C09129=1221.568,302.817,-67.481,-176.404,6.935,148.235
C09130=1221.564,303.066,-67.511,-176.401,6.937,148.235
C09131=1221.559,303.313,-67.540,-176.399,6.940,148.235
C09132=1221.555,303.561,-67.570,-176.397,6.942,148.235
C09133=1221.551,303.809,-67.599,-176.395,6.944,148.235
C09134=1221.546,304.058,-67.629,-176.392,6.947,148.235
C09135=1221.542,304.306,-67.659,-176.390,6.950,148.235
C09136=1221.538,304.554,-67.688,-176.387,6.953,148.235
C09137=1221.533,304.803,-67.718,-176.385,6.955,148.235
C09138=1221.529,305.051,-67.747,-176.383,6.957,148.235
C09139=1221.525,305.299,-67.778,-176.380,6.960,148.235
C09140=1221.520,305.547,-67.807,-176.378,6.962,148.235
C09141=1221.516,305.795,-67.837,-176.376,6.965,148.235
C09142=1221.512,306.044,-67.866,-176.373,6.968,148.235
C09143=1221.508,306.291,-67.896,-176.371,6.970,148.235
C09144=1221.503,306.540,-67.926,-176.369,6.973,148.235
C09145=1221.499,306.788,-67.956,-176.366,6.975,148.235
C09146=1221.495,307.036,-67.985,-176.364,6.977,148.234
C09147=1221.491,307.284,-68.016,-176.362,6.980,148.234
C09148=1221.486,307.533,-68.046,-176.360,6.983,148.234
C09149=1221.482,307.781,-68.075,-176.357,6.986,148.234
C09150=1221.478,308.029,-68.104,-176.355,6.988,148.234
C09151=1221.473,308.277,-68.135,-176.353,6.990,148.234
C09152=1221.469,308.525,-68.165,-176.350,6.993,148.234
C09153=1221.465,308.774,-68.194,-176.348,6.995,148.234
C09154=1221.460,309.022,-68.225,-176.346,6.998,148.234
C09155=1221.456,309.270,-68.254,-176.343,7.001,148.234
C09156=1221.452,309.517,-68.285,-176.341,7.003,148.234
C09157=1221.447,309.766,-68.315,-176.338,7.006,148.234
C09158=1221.443,310.014,-68.344,-176.336,7.008,148.234
C09159=1221.439,310.262,-68.374,-176.334,7.010,148.234
C09160=1221.434,310.511,-68.404,-176.332,7.013,148.234
C09161=1221.430,310.758,-68.434,-176.329,7.016,148.234
C09162=1221.426,311.006,-68.464,-176.327,7.019,148.234
C09163=1221.422,311.256,-68.494,-176.325,7.021,148.234
C09164=1221.418,311.503,-68.524,-176.323,7.023,148.234
C09165=1221.413,311.752,-68.554,-176.320,7.026,148.234
C09166=1221.409,312.000,-68.585,-176.318,7.028,148.234
C09167=1221.405,312.248,-68.614,-176.316,7.032,148.234
C09168=1221.400,312.496,-68.645,-176.313,7.034,148.234
C09169=1221.396,312.743,-68.675,-176.311,7.036,148.234
C09170=1221.391,312.992,-68.705,-176.309,7.039,148.234
C09171=1221.388,313.240,-68.735,-176.307,7.041,148.234
C09172=1221.383,313.488,-68.765,-176.304,7.044,148.234
C09173=1221.379,313.737,-68.796,-176.302,7.047,148.234
C09174=1221.375,313.985,-68.826,-176.300,7.049,148.234
C09175=1221.371,314.233,-68.856,-176.298,7.052,148.234
C09176=1221.367,314.480,-68.886,-176.295,7.054,148.234
C09177=1221.362,314.729,-68.916,-176.293,7.058,148.234
C09178=1221.357,315.005,-68.951,-176.291,7.060,148.234
C09179=1221.353,315.281,-68.984,-176.288,7.063,148.234
C09180=1221.348,315.557,-69.018,-176.285,7.066,148.234
C09181=1221.343,315.832,-69.050,-176.283,7.069,148.234
C09182=1221.339,316.081,-69.082,-176.281,7.071,148.234
C09183=1221.334,316.329,-69.112,-176.278,7.074,148.234
C09184=1221.330,316.577,-69.142,-176.276,7.077,148.234
C09185=1221.326,316.825,-69.173,-176.274,7.079,148.234
C09186=1221.322,317.073,-69.203,-176.271,7.082,148.234
C09187=1221.317,317.321,-69.233,-176.269,7.084,148.234
C09188=1221.313,317.570,-69.263,-176.267,7.087,148.234
C09189=1221.309,317.818,-69.294,-176.265,7.090,148.234
C09190=1221.305,318.065,-69.324,-176.262,7.093,148.234
C09191=1221.300,318.313,-69.355,-176.260,7.095,148.234
C09192=1221.295,318.562,-69.385,-176.258,7.097,148.234
C09193=1221.292,318.810,-69.416,-176.256,7.101,148.234
C09194=1221.288,319.058,-69.446,-176.254,7.103,148.234
C09195=1221.283,319.306,-69.477,-176.251,7.106,148.234
C09196=1221.279,319.554,-69.507,-176.249,7.108,148.234
C09197=1221.275,319.802,-69.538,-176.247,7.111,148.234
C09198=1221.271,320.051,-69.568,-176.245,7.114,148.234
C09199=1221.266,320.298,-69.599,-176.243,7.116,148.234
C09200=1221.262,320.546,-69.629,-176.240,7.119,148.234
C09201=1221.258,320.795,-69.660,-176.238,7.121,148.234
C09202=1221.254,321.043,-69.691,-176.236,7.124,148.234
C09203=1221.249,321.291,-69.721,-176.234,7.127,148.234
C09204=1221.245,321.538,-69.752,-176.232,7.129,148.234
C09205=1221.241,321.787,-69.783,-176.229,7.132,148.235
C09206=1221.237,322.035,-69.813,-176.227,7.134,148.234
C09207=1221.232,322.283,-69.844,-176.225,7.138,148.234
C09208=1221.228,322.531,-69.874,-176.223,7.140,148.235
C09209=1221.224,322.779,-69.906,-176.221,7.142,148.235
C09210=1221.220,323.027,-69.936,-176.218,7.145,148.235
C09211=1221.216,323.275,-69.966,-176.217,7.148,148.235
C09212=1221.212,323.524,-69.998,-176.214,7.151,148.235
C09213=1221.207,323.771,-70.028,-176.212,7.153,148.235
C09214=1221.202,324.019,-70.059,-176.210,7.156,148.235
C09215=1221.199,324.268,-70.090,-176.207,7.159,148.235
C09216=1221.195,324.516,-70.120,-176.205,7.161,148.235
C09217=1221.190,324.764,-70.151,-176.203,7.164,148.235
C09218=1221.186,325.012,-70.182,-176.201,7.166,148.235
C09219=1221.181,325.260,-70.213,-176.198,7.170,148.235
C09220=1221.178,325.507,-70.244,-176.197,7.172,148.235
C09221=1221.174,325.756,-70.275,-176.195,7.174,148.235
C09222=1221.169,326.004,-70.306,-176.192,7.178,148.235
C09223=1221.165,326.252,-70.337,-176.190,7.180,148.235
C09224=1221.161,326.501,-70.368,-176.188,7.183,148.235
C09225=1221.157,326.748,-70.398,-176.186,7.185,148.236
C09226=1221.152,326.996,-70.429,-176.184,7.188,148.235
C09227=1221.148,327.244,-70.461,-176.182,7.191,148.236
C09228=1221.144,327.492,-70.491,-176.180,7.193,148.236
C09229=1221.139,327.740,-70.522,-176.177,7.196,148.236
C09230=1221.135,327.989,-70.553,-176.175,7.199,148.236
C09231=1221.131,328.236,-70.585,-176.173,7.202,148.236
C09232=1221.127,328.485,-70.616,-176.171,7.204,148.236
C09233=1221.122,328.733,-70.647,-176.169,7.207,148.236
C09234=1221.119,328.980,-70.677,-176.167,7.210,148.236
C09235=1221.115,329.228,-70.709,-176.165,7.212,148.236
C09236=1221.110,329.476,-70.739,-176.163,7.216,148.236
C09237=1221.105,329.724,-70.770,-176.160,7.218,148.236
C09238=1221.102,329.972,-70.802,-176.159,7.220,148.237
C09239=1221.097,330.220,-70.833,-176.156,7.223,148.237
C09240=1221.093,330.469,-70.864,-176.154,7.226,148.237
C09241=1221.089,330.716,-70.895,-176.152,7.229,148.237
C09242=1221.085,330.965,-70.926,-176.150,7.231,148.237
C09243=1221.080,331.212,-70.958,-176.148,7.234,148.237
C09244=1221.076,331.460,-70.989,-176.146,7.237,148.237
C09245=1221.072,331.709,-71.020,-176.144,7.239,148.237
C09246=1221.067,331.956,-71.051,-176.142,7.243,148.237
C09247=1221.063,332.205,-71.082,-176.139,7.245,148.237
C09248=1221.059,332.452,-71.114,-176.137,7.248,148.237
C09249=1221.055,332.701,-71.145,-176.135,7.250,148.237
C09250=1221.051,332.948,-71.177,-176.134,7.253,148.238
C09251=1221.047,333.197,-71.208,-176.131,7.256,148.238
C09252=1221.042,333.444,-71.239,-176.129,7.258,148.238
C09253=1221.038,333.693,-71.270,-176.127,7.262,148.238
C09254=1221.034,333.940,-71.302,-176.125,7.264,148.238
C09255=1221.030,334.188,-71.333,-176.123,7.267,148.238
C09256=1221.026,334.436,-71.364,-176.121,7.270,148.238
C09257=1221.021,334.684,-71.395,-176.119,7.272,148.238
C09258=1221.017,334.933,-71.428,-176.117,7.276,148.239
C09259=1221.012,335.181,-71.458,-176.115,7.278,148.238
C09260=1221.008,335.429,-71.490,-176.113,7.280,148.239
C09261=1221.004,335.677,-71.521,-176.111,7.284,148.239
C09262=1221.000,335.925,-71.553,-176.109,7.286,148.239
C09263=1220.996,336.172,-71.584,-176.107,7.289,148.239
C09264=1220.992,336.421,-71.615,-176.105,7.291,148.239
C09265=1220.988,336.669,-71.647,-176.103,7.294,148.239
C09266=1220.984,336.916,-71.679,-176.101,7.297,148.239
C09267=1220.979,337.165,-71.710,-176.099,7.300,148.239
C09268=1220.975,337.412,-71.742,-176.096,7.303,148.240
C09269=1220.971,337.660,-71.774,-176.095,7.305,148.240
C09270=1220.966,337.908,-71.805,-176.093,7.308,148.240
C09271=1220.963,338.156,-71.836,-176.090,7.311,148.240
C09272=1220.958,338.404,-71.868,-176.089,7.314,148.240
C09273=1220.954,338.653,-71.900,-176.087,7.317,148.240
C09274=1220.949,338.900,-71.931,-176.085,7.319,148.240
C09275=1220.946,339.148,-71.963,-176.083,7.322,148.241
C09276=1220.942,339.396,-71.995,-176.081,7.325,148.241
C09277=1220.937,339.644,-72.026,-176.079,7.328,148.241
C09278=1220.933,339.892,-72.058,-176.076,7.331,148.241
C09279=1220.929,340.140,-72.089,-176.075,7.333,148.241
C09280=1220.925,340.388,-72.121,-176.073,7.336,148.241
C09281=1220.921,340.635,-72.153,-176.071,7.339,148.242
C09282=1220.915,340.913,-72.188,-176.068,7.342,148.242
C09283=1220.911,341.191,-72.224,-176.067,7.345,148.242
C09284=1220.907,341.469,-72.259,-176.064,7.348,148.242
C09285=1220.901,341.747,-72.295,-176.062,7.351,148.242
C09286=1220.897,341.995,-72.327,-176.060,7.353,148.242
C09287=1220.894,342.243,-72.359,-176.058,7.357,148.242
C09288=1220.889,342.491,-72.391,-176.056,7.359,148.243
C09289=1220.885,342.739,-72.423,-176.055,7.362,148.243
C09290=1220.881,342.986,-72.454,-176.053,7.365,148.243
C09291=1220.876,343.234,-72.486,-176.050,7.367,148.243
C09292=1220.872,343.483,-72.518,-176.048,7.371,148.243
C09293=1220.868,343.730,-72.549,-176.047,7.373,148.243
C09294=1220.864,343.979,-72.582,-176.045,7.376,148.244
C09295=1220.860,344.227,-72.613,-176.043,7.379,148.244
C09296=1220.856,344.474,-72.645,-176.041,7.382,148.244
C09297=1220.851,344.723,-72.677,-176.040,7.384,148.244
C09298=1220.847,344.971,-72.709,-176.037,7.388,148.244
C09299=1220.842,345.218,-72.741,-176.035,7.390,148.244
C09300=1220.839,345.466,-72.773,-176.033,7.393,148.245
C09301=1220.835,345.714,-72.805,-176.031,7.396,148.245
C09302=1220.830,345.962,-72.837,-176.030,7.398,148.245
C09303=1220.826,346.210,-72.869,-176.028,7.402,148.245
C09304=1220.822,346.458,-72.902,-176.026,7.404,148.245
C09305=1220.818,346.705,-72.933,-176.024,7.407,148.245
C09306=1220.814,346.953,-72.965,-176.022,7.410,148.246
C09307=1220.810,347.201,-72.998,-176.020,7.413,148.246
C09308=1220.805,347.449,-73.029,-176.019,7.415,148.246
C09309=1220.801,347.697,-73.062,-176.017,7.418,148.246
C09310=1220.797,347.945,-73.094,-176.015,7.421,148.246
C09311=1220.792,348.193,-73.126,-176.013,7.424,148.247
C09312=1220.788,348.441,-73.157,-176.011,7.427,148.247
C09313=1220.784,348.689,-73.191,-176.010,7.429,148.247
C09314=1220.781,348.937,-73.222,-176.007,7.433,148.247
C09315=1220.775,349.184,-73.254,-176.006,7.435,148.247
C09316=1220.772,349.432,-73.286,-176.004,7.438,148.248
C09317=1220.767,349.681,-73.319,-176.002,7.441,148.248
C09318=1220.764,349.928,-73.351,-176.000,7.444,148.248
C09319=1220.759,350.176,-73.383,-175.999,7.446,148.248
C09320=1220.755,350.424,-73.415,-175.996,7.450,148.248
C09321=1220.751,350.672,-73.448,-175.995,7.452,148.249
C09322=1220.747,350.920,-73.480,-175.993,7.455,148.249
C09323=1220.742,351.167,-73.512,-175.991,7.458,148.249
C09324=1220.739,351.415,-73.544,-175.989,7.460,148.249
C09325=1220.734,351.664,-73.577,-175.988,7.463,148.249
C09326=1220.730,351.911,-73.610,-175.986,7.466,148.250
C09327=1220.726,352.159,-73.641,-175.984,7.469,148.250
C09328=1220.721,352.407,-73.674,-175.983,7.472,148.250
C09329=1220.718,352.654,-73.706,-175.981,7.475,148.250
C09330=1220.713,352.903,-73.739,-175.979,7.478,148.251
C09331=1220.710,353.151,-73.771,-175.977,7.480,148.251
C09332=1220.705,353.398,-73.803,-175.975,7.483,148.251
C09333=1220.700,353.646,-73.836,-175.973,7.486,148.251
C09334=1220.697,353.894,-73.868,-175.972,7.489,148.252
C09335=1220.693,354.142,-73.901,-175.970,7.492,148.252
C09336=1220.688,354.390,-73.933,-175.968,7.495,148.252
C09337=1220.684,354.637,-73.965,-175.967,7.497,148.252
C09338=1220.680,354.885,-73.998,-175.965,7.500,148.252
C09339=1220.676,355.133,-74.030,-175.963,7.503,148.253
C09340=1220.672,355.381,-74.063,-175.962,7.506,148.253
C09341=1220.667,355.629,-74.095,-175.960,7.508,148.253
C09342=1220.664,355.877,-74.128,-175.958,7.512,148.253
C09343=1220.659,356.125,-74.160,-175.956,7.514,148.254
C09344=1220.655,356.372,-74.193,-175.955,7.517,148.254
C09345=1220.651,356.620,-74.225,-175.953,7.521,148.254
C09346=1220.647,356.868,-74.258,-175.951,7.523,148.254
C09347=1220.643,357.116,-74.291,-175.950,7.526,148.255
C09348=1220.638,357.364,-74.324,-175.949,7.528,148.255
C09349=1220.635,357.612,-74.356,-175.946,7.532,148.255
C09350=1220.630,357.859,-74.388,-175.945,7.534,148.255
C09351=1220.626,358.107,-74.421,-175.943,7.537,148.256
C09352=1220.622,358.355,-74.453,-175.941,7.540,148.256
C09353=1220.618,358.603,-74.486,-175.940,7.543,148.256
C09354=1220.614,358.851,-74.519,-175.938,7.546,148.257
C09355=1220.609,359.099,-74.552,-175.937,7.548,148.257
C09356=1220.606,359.346,-74.585,-175.935,7.552,148.257
C09357=1220.602,359.595,-74.617,-175.933,7.554,148.257
C09358=1220.597,359.842,-74.650,-175.932,7.557,148.258
C09359=1220.592,360.090,-74.682,-175.930,7.560,148.258
C09360=1220.588,360.338,-74.715,-175.928,7.563,148.258
C09361=1220.585,360.585,-74.748,-175.927,7.566,148.258
C09362=1220.580,360.833,-74.780,-175.925,7.568,148.259
C09363=1220.576,361.081,-74.814,-175.924,7.571,148.259
C09364=1220.572,361.329,-74.847,-175.922,7.574,148.259
C09365=1220.568,361.577,-74.880,-175.921,7.577,148.260
C09366=1220.564,361.825,-74.912,-175.919,7.580,148.260
C09367=1220.560,362.072,-74.945,-175.918,7.583,148.260
C09368=1220.556,362.320,-74.978,-175.916,7.586,148.261
C09369=1220.552,362.568,-75.011,-175.914,7.588,148.261
C09370=1220.547,362.816,-75.044,-175.913,7.591,148.261
C09371=1220.543,363.064,-75.077,-175.911,7.594,148.261
C09372=1220.540,363.311,-75.109,-175.910,7.597,148.262
C09373=1220.536,363.559,-75.143,-175.908,7.600,148.262
C09374=1220.531,363.807,-75.175,-175.907,7.603,148.262
C09375=1220.527,364.054,-75.208,-175.905,7.605,148.262
C09376=1220.522,364.302,-75.241,-175.904,7.608,148.263
C09377=1220.518,364.550,-75.274,-175.903,7.611,148.263
C09378=1220.514,364.798,-75.307,-175.900,7.614,148.264
C09379=1220.510,365.046,-75.340,-175.899,7.617,148.264
C09380=1220.506,365.293,-75.372,-175.898,7.620,148.264
C09381=1220.502,365.541,-75.405,-175.896,7.622,148.264
C09382=1220.498,365.789,-75.439,-175.895,7.625,148.265
C09383=1220.494,366.037,-75.472,-175.893,7.629,148.265
C09384=1220.490,366.284,-75.505,-175.891,7.631,148.265
C09385=1220.486,366.532,-75.538,-175.890,7.634,148.266
C09386=1220.481,366.813,-75.575,-175.889,7.637,148.266
C09387=1220.477,367.093,-75.613,-175.887,7.640,148.266
C09388=1220.472,367.372,-75.650,-175.885,7.644,148.267
C09389=1220.468,367.652,-75.688,-175.884,7.647,148.267
C09390=1220.463,367.900,-75.720,-175.883,7.649,148.268
C09391=1220.459,368.148,-75.753,-175.881,7.652,148.268
C09392=1220.455,368.396,-75.787,-175.879,7.656,148.268
C09393=1220.451,368.643,-75.820,-175.878,7.658,148.269
C09394=1220.447,368.891,-75.853,-175.877,7.661,148.269
C09395=1220.442,369.139,-75.886,-175.875,7.664,148.269
C09396=1220.438,369.386,-75.919,-175.874,7.667,148.270
C09397=1220.434,369.634,-75.952,-175.873,7.669,148.270
C09398=1220.430,369.882,-75.985,-175.871,7.672,148.270
C09399=1220.426,370.130,-76.019,-175.870,7.675,148.271
C09400=1220.422,370.377,-76.053,-175.869,7.678,148.271
C09401=1220.418,370.624,-76.086,-175.867,7.680,148.271
C09402=1220.414,370.872,-76.119,-175.866,7.683,148.272
C09403=1220.410,371.120,-76.152,-175.865,7.687,148.272
C09404=1220.405,371.368,-76.185,-175.863,7.689,148.272
C09405=1220.401,371.616,-76.219,-175.862,7.692,148.273
C09406=1220.397,371.864,-76.252,-175.861,7.695,148.273
C09407=1220.393,372.112,-76.286,-175.859,7.698,148.273
C09408=1220.389,372.360,-76.319,-175.858,7.700,148.274
C09409=1220.385,372.607,-76.352,-175.857,7.703,148.274
C09410=1220.381,372.854,-76.386,-175.856,7.706,148.275
C09411=1220.377,373.102,-76.419,-175.854,7.709,148.275
C09412=1220.373,373.350,-76.452,-175.853,7.711,148.275
C09413=1220.368,373.598,-76.485,-175.852,7.714,148.276
C09414=1220.364,373.845,-76.518,-175.851,7.717,148.276
C09415=1220.359,374.093,-76.552,-175.849,7.720,148.276
C09416=1220.356,374.341,-76.586,-175.848,7.723,148.277
C09417=1220.352,374.589,-76.620,-175.847,7.726,148.277
C09418=1220.348,374.837,-76.653,-175.846,7.728,148.277
C09419=1220.344,375.084,-76.686,-175.845,7.731,148.278
C09420=1220.340,375.332,-76.719,-175.843,7.734,148.278
C09421=1220.336,375.579,-76.753,-175.842,7.736,148.278
C09422=1220.331,375.827,-76.787,-175.841,7.739,148.279
C09423=1220.327,376.075,-76.820,-175.840,7.742,148.279
C09424=1220.323,376.323,-76.853,-175.838,7.745,148.280
C09425=1220.319,376.571,-76.887,-175.837,7.748,148.280
C09426=1220.315,376.818,-76.920,-175.836,7.751,148.280
C09427=1220.311,377.066,-76.953,-175.835,7.753,148.281
C09428=1220.307,377.313,-76.988,-175.834,7.755,148.281
C09429=1220.302,377.561,-77.021,-175.833,7.758,148.282
C09430=1220.298,377.809,-77.054,-175.832,7.761,148.282
C09431=1220.295,378.057,-77.088,-175.831,7.764,148.282
C09432=1220.291,378.304,-77.122,-175.829,7.767,148.283
C09433=1220.286,378.552,-77.155,-175.828,7.769,148.283
C09434=1220.282,378.800,-77.189,-175.827,7.772,148.284
C09435=1220.278,379.047,-77.222,-175.826,7.775,148.284
C09436=1220.274,379.295,-77.256,-175.825,7.778,148.284
C09437=1220.270,379.543,-77.290,-175.824,7.781,148.285
C09438=1220.266,379.791,-77.324,-175.823,7.783,148.285
C09439=1220.262,380.039,-77.357,-175.822,7.786,148.285
C09440=1220.258,380.286,-77.391,-175.821,7.789,148.286
C09441=1220.253,380.534,-77.424,-175.820,7.791,148.286
C09442=1220.249,380.781,-77.458,-175.819,7.794,148.287
C09443=1220.246,381.029,-77.492,-175.817,7.797,148.287
C09444=1220.241,381.277,-77.525,-175.816,7.800,148.288
C09445=1220.237,381.524,-77.559,-175.816,7.802,148.288
C09446=1220.233,381.772,-77.593,-175.814,7.805,148.288
C09447=1220.229,382.019,-77.626,-175.813,7.808,148.289
C09448=1220.225,382.268,-77.660,-175.812,7.810,148.289
C09449=1220.221,382.515,-77.694,-175.811,7.813,148.290
C09450=1220.217,382.763,-77.728,-175.811,7.815,148.290
C09451=1220.212,383.010,-77.762,-175.810,7.818,148.291
C09452=1220.209,383.259,-77.796,-175.808,7.821,148.291
C09453=1220.205,383.506,-77.829,-175.807,7.824,148.291
C09454=1220.200,383.754,-77.863,-175.807,7.826,148.292
C09455=1220.196,384.001,-77.897,-175.805,7.829,148.292
C09456=1220.192,384.249,-77.930,-175.805,7.832,148.293
C09457=1220.188,384.497,-77.965,-175.803,7.835,148.293
C09458=1220.184,384.745,-77.998,-175.802,7.837,148.293
C09459=1220.180,384.992,-78.032,-175.802,7.839,148.294
C09460=1220.175,385.240,-78.066,-175.800,7.842,148.294
C09461=1220.172,385.487,-78.100,-175.800,7.845,148.295
C09462=1220.168,385.735,-78.134,-175.799,7.847,148.295
C09463=1220.163,385.983,-78.168,-175.798,7.850,148.296
C09464=1220.159,386.230,-78.202,-175.797,7.853,148.296
C09465=1220.155,386.478,-78.236,-175.796,7.856,148.297
C09466=1220.151,386.726,-78.269,-175.795,7.858,148.297
C09467=1220.147,386.973,-78.303,-175.794,7.861,148.297
C09468=1220.142,387.221,-78.337,-175.793,7.864,148.298
C09469=1220.139,387.469,-78.371,-175.793,7.866,148.298
C09470=1220.134,387.717,-78.405,-175.792,7.869,148.299
C09471=1220.131,387.964,-78.439,-175.790,7.872,148.299
C09472=1220.127,388.211,-78.473,-175.790,7.874,148.299
C09473=1220.122,388.460,-78.507,-175.789,7.877,148.300
C09474=1220.119,388.707,-78.541,-175.788,7.880,148.300
C09475=1220.114,388.954,-78.575,-175.787,7.881,148.301
C09476=1220.111,389.202,-78.609,-175.786,7.884,148.301
C09477=1220.106,389.450,-78.643,-175.785,7.887,148.302
C09478=1220.102,389.697,-78.677,-175.785,7.889,148.302
C09479=1220.099,389.945,-78.711,-175.783,7.892,148.302
C09480=1220.094,390.193,-78.745,-175.783,7.894,148.303
C09481=1220.090,390.440,-78.779,-175.782,7.897,148.303
C09482=1220.086,390.687,-78.813,-175.781,7.900,148.304
C09483=1220.082,390.936,-78.847,-175.781,7.902,148.304
C09484=1220.077,391.183,-78.881,-175.780,7.905,148.305
C09485=1220.074,391.430,-78.915,-175.779,7.907,148.305
C09486=1220.070,391.678,-78.950,-175.778,7.910,148.306
C09487=1220.066,391.926,-78.983,-175.777,7.913,148.306
C09488=1220.061,392.174,-79.018,-175.776,7.915,148.306
C09489=1220.058,392.421,-79.052,-175.776,7.918,148.307
C09490=1220.053,392.703,-79.091,-175.774,7.921,148.307
C09491=1220.048,392.985,-79.130,-175.774,7.923,148.308
C09492=1220.044,393.267,-79.169,-175.773,7.926,148.308
C09493=1220.039,393.549,-79.207,-175.772,7.929,148.309
C09494=1220.035,393.796,-79.242,-175.771,7.932,148.309
C09495=1220.031,394.044,-79.276,-175.771,7.934,148.310
C09496=1220.027,394.291,-79.310,-175.770,7.937,148.310
C09497=1220.023,394.539,-79.344,-175.769,7.939,148.311
C09498=1220.019,394.787,-79.378,-175.768,7.942,148.311
C09499=1220.015,395.034,-79.412,-175.768,7.944,148.312
C09500=1220.010,395.282,-79.447,-175.767,7.947,148.312
C09501=1220.007,395.529,-79.481,-175.766,7.949,148.312
C09502=1220.002,395.777,-79.515,-175.765,7.952,148.313
C09503=1219.998,396.024,-79.550,-175.765,7.954,148.313
C09504=1219.995,396.272,-79.584,-175.764,7.957,148.314
C09505=1219.990,396.520,-79.618,-175.763,7.959,148.314
C09506=1219.986,396.767,-79.652,-175.763,7.961,148.315
C09507=1219.982,397.015,-79.687,-175.762,7.964,148.315
C09508=1219.978,397.262,-79.720,-175.762,7.967,148.316
C09509=1219.974,397.511,-79.755,-175.760,7.969,148.316
C09510=1219.970,397.758,-79.790,-175.760,7.972,148.317
C09511=1219.966,398.005,-79.824,-175.759,7.974,148.317
C09512=1219.962,398.253,-79.858,-175.758,7.976,148.317
C09513=1219.958,398.500,-79.892,-175.758,7.979,148.318
C09514=1219.953,398.748,-79.927,-175.757,7.982,148.318
C09515=1219.949,398.996,-79.962,-175.757,7.984,148.319
C09516=1219.946,399.243,-79.995,-175.756,7.987,148.319
C09517=1219.942,399.491,-80.030,-175.755,7.989,148.319
C09518=1219.937,399.739,-80.065,-175.755,7.991,148.320
C09519=1219.933,399.986,-80.099,-175.754,7.994,148.320
C09520=1219.929,400.234,-80.134,-175.753,7.996,148.321
C09521=1219.925,400.481,-80.167,-175.753,7.998,148.321
C09522=1219.921,400.729,-80.202,-175.752,8.001,148.322
C09523=1219.917,400.976,-80.237,-175.751,8.003,148.322
C09524=1219.913,401.224,-80.271,-175.751,8.006,148.323
C09525=1219.909,401.472,-80.305,-175.750,8.008,148.323
C09526=1219.904,401.719,-80.340,-175.749,8.010,148.324
C09527=1219.901,401.967,-80.374,-175.749,8.013,148.324
C09528=1219.897,402.214,-80.409,-175.748,8.015,148.324
C09529=1219.893,402.462,-80.443,-175.748,8.017,148.325
C09530=1219.889,402.710,-80.477,-175.747,8.019,148.325
C09531=1219.884,402.957,-80.512,-175.746,8.023,148.326
C09532=1219.880,403.205,-80.547,-175.746,8.024,148.326
C09533=1219.877,403.452,-80.580,-175.746,8.027,148.327
C09534=1219.873,403.700,-80.615,-175.744,8.030,148.327
C09535=1219.868,403.948,-80.650,-175.744,8.032,148.328
C09536=1219.865,404.196,-80.684,-175.744,8.034,148.328
C09537=1219.860,404.443,-80.718,-175.743,8.036,148.328
C09538=1219.856,404.690,-80.753,-175.742,8.039,148.329
C09539=1219.852,404.938,-80.788,-175.742,8.041,148.329
C09540=1219.848,405.185,-80.822,-175.741,8.043,148.330
C09541=1219.844,405.433,-80.857,-175.741,8.045,148.330
C09542=1219.840,405.681,-80.892,-175.740,8.048,148.331
C09543=1219.836,405.928,-80.926,-175.739,8.050,148.331
C09544=1219.832,406.176,-80.960,-175.739,8.052,148.332
C09545=1219.828,406.424,-80.995,-175.739,8.054,148.332
C09546=1219.823,406.671,-81.030,-175.737,8.057,148.332
C09547=1219.820,406.918,-81.065,-175.737,8.060,148.333
C09548=1219.816,407.166,-81.099,-175.736,8.062,148.333
C09549=1219.811,407.413,-81.133,-175.736,8.064,148.334
C09550=1219.808,407.661,-81.168,-175.736,8.066,148.334
C09551=1219.803,407.909,-81.202,-175.735,8.069,148.335
C09552=1219.799,408.157,-81.237,-175.734,8.071,148.335
C09553=1219.795,408.403,-81.272,-175.734,8.073,148.336
C09554=1219.791,408.652,-81.307,-175.733,8.075,148.336
C09555=1219.787,408.899,-81.341,-175.733,8.077,148.337
C09556=1219.783,409.147,-81.376,-175.732,8.080,148.337
C09557=1219.779,409.394,-81.411,-175.732,8.082,148.338
C09558=1219.775,409.642,-81.446,-175.731,8.084,148.338
C09559=1219.771,409.889,-81.480,-175.731,8.086,148.338
C09560=1219.767,410.137,-81.514,-175.730,8.089,148.339
C09561=1219.763,410.384,-81.549,-175.730,8.091,148.339
C09562=1219.759,410.632,-81.584,-175.730,8.093,148.340
C09563=1219.755,410.879,-81.618,-175.728,8.096,148.340
C09564=1219.751,411.127,-81.653,-175.728,8.098,148.341
C09565=1219.747,411.375,-81.688,-175.728,8.100,148.341
C09566=1219.743,411.622,-81.723,-175.727,8.102,148.341
C09567=1219.738,411.869,-81.758,-175.727,8.104,148.342
C09568=1219.735,412.117,-81.792,-175.726,8.106,148.342
C09569=1219.731,412.364,-81.827,-175.726,8.108,148.343
C09570=1219.727,412.612,-81.862,-175.725,8.110,148.343
C09571=1219.722,412.860,-81.896,-175.724,8.114,148.344
C09572=1219.718,413.108,-81.931,-175.724,8.116,148.344
C09573=1219.714,413.355,-81.966,-175.724,8.118,148.344
C09574=1219.711,413.602,-82.001,-175.723,8.120,148.345
C09575=1219.706,413.850,-82.035,-175.723,8.122,148.345
C09576=1219.703,414.097,-82.071,-175.722,8.124,148.346
C09577=1219.698,414.345,-82.105,-175.721,8.126,148.346
C09578=1219.694,414.593,-82.140,-175.721,8.128,148.347
C09579=1219.690,414.840,-82.175,-175.721,8.130,148.347
C09580=1219.687,415.087,-82.209,-175.720,8.133,148.347
C09581=1219.683,415.336,-82.244,-175.720,8.134,148.348
C09582=1219.679,415.554,-82.276,-175.719,8.136,148.348
C09583=1219.675,415.774,-82.306,-175.719,8.139,148.349
C09584=1219.672,415.994,-82.337,-175.718,8.141,148.349
C09585=1219.668,416.213,-82.369,-175.718,8.143,148.349
C09586=1219.664,416.432,-82.399,-175.717,8.145,148.350
C09587=1219.661,416.652,-82.430,-175.717,8.146,148.350
C09588=1219.658,416.871,-82.461,-175.717,8.148,148.350
C09589=1219.658,417.090,-82.491,-175.716,8.150,148.351
C09590=1219.236,417.091,-82.526,-175.719,8.161,148.355
C09591=1219.236,416.870,-82.495,-175.720,8.159,148.354
C09592=1219.239,416.649,-82.465,-175.720,8.156,148.354
C09593=1219.242,416.428,-82.433,-175.720,8.155,148.353
C09594=1219.246,416.208,-82.402,-175.721,8.153,148.353
C09595=1219.250,415.986,-82.371,-175.722,8.151,148.353
C09596=1219.253,415.766,-82.339,-175.722,8.149,148.352
C09597=1219.257,415.545,-82.309,-175.723,8.147,148.352
C09598=1219.260,415.324,-82.278,-175.723,8.145,148.352
C09599=1219.265,415.077,-82.243,-175.723,8.143,148.351
C09600=1219.268,414.829,-82.208,-175.724,8.141,148.351
C09601=1219.273,414.582,-82.173,-175.724,8.139,148.350
C09602=1219.277,414.334,-82.138,-175.725,8.137,148.350
C09603=1219.281,414.087,-82.103,-175.726,8.135,148.349
C09604=1219.285,413.839,-82.068,-175.726,8.132,148.349
C09605=1219.289,413.592,-82.035,-175.726,8.130,148.349
C09606=1219.292,413.344,-81.999,-175.727,8.128,148.348
C09607=1219.297,413.097,-81.965,-175.727,8.126,148.348
C09608=1219.301,412.849,-81.930,-175.727,8.124,148.347
C09609=1219.305,412.602,-81.895,-175.729,8.121,148.347
C09610=1219.309,412.354,-81.860,-175.729,8.119,148.346
C09611=1219.313,412.107,-81.826,-175.729,8.117,148.346
C09612=1219.317,411.859,-81.790,-175.730,8.115,148.346
C09613=1219.321,411.612,-81.756,-175.730,8.113,148.345
C09614=1219.325,411.364,-81.721,-175.731,8.111,148.345
C09615=1219.330,411.116,-81.687,-175.731,8.108,148.344
C09616=1219.333,410.869,-81.652,-175.732,8.106,148.344
C09617=1219.337,410.622,-81.617,-175.733,8.103,148.343
C09618=1219.341,410.374,-81.582,-175.733,8.101,148.343
C09619=1219.346,410.126,-81.548,-175.733,8.099,148.342
C09620=1219.350,409.879,-81.512,-175.734,8.097,148.342
C09621=1219.353,409.632,-81.478,-175.734,8.095,148.341
C09622=1219.357,409.383,-81.444,-175.735,8.093,148.341
C09623=1219.362,409.136,-81.409,-175.735,8.091,148.341
C09624=1219.366,408.888,-81.374,-175.736,8.088,148.340
C09625=1219.369,408.641,-81.340,-175.737,8.086,148.340
C09626=1219.373,408.393,-81.305,-175.737,8.083,148.339
C09627=1219.378,408.146,-81.270,-175.738,8.081,148.339
C09628=1219.382,407.898,-81.236,-175.738,8.079,148.338
C09629=1219.385,407.651,-81.201,-175.739,8.076,148.338
C09630=1219.389,407.403,-81.166,-175.739,8.074,148.337
C09631=1219.394,407.156,-81.132,-175.740,8.072,148.337
C09632=1219.398,406.908,-81.097,-175.740,8.070,148.337
C09633=1219.402,406.660,-81.063,-175.741,8.068,148.336
C09634=1219.406,406.412,-81.028,-175.742,8.065,148.336
C09635=1219.410,406.166,-80.993,-175.742,8.063,148.335
C09636=1219.414,405.917,-80.958,-175.742,8.061,148.335
C09637=1219.418,405.670,-80.924,-175.743,8.059,148.334
C09638=1219.422,405.422,-80.889,-175.744,8.055,148.334
C09639=1219.426,405.175,-80.855,-175.744,8.053,148.333
C09640=1219.431,404.927,-80.820,-175.745,8.052,148.333
C09641=1219.434,404.680,-80.786,-175.745,8.049,148.333
C09642=1219.438,404.433,-80.751,-175.746,8.046,148.332
C09643=1219.442,404.185,-80.716,-175.747,8.044,148.332
C09644=1219.446,403.938,-80.682,-175.747,8.042,148.331
C09645=1219.450,403.689,-80.648,-175.747,8.040,148.331
C09646=1219.455,403.442,-80.613,-175.749,8.037,148.330
C09647=1219.458,403.194,-80.579,-175.749,8.035,148.330
C09648=1219.463,402.947,-80.544,-175.749,8.033,148.330
C09649=1219.467,402.699,-80.510,-175.750,8.030,148.329
C09650=1219.470,402.452,-80.476,-175.751,8.028,148.329
C09651=1219.475,402.204,-80.441,-175.751,8.025,148.328
C09652=1219.479,401.956,-80.406,-175.752,8.024,148.328
C09653=1219.483,401.709,-80.372,-175.753,8.021,148.327
C09654=1219.487,401.461,-80.338,-175.753,8.018,148.327
C09655=1219.491,401.213,-80.303,-175.754,8.016,148.326
C09656=1219.495,400.966,-80.269,-175.754,8.013,148.326
C09657=1219.499,400.718,-80.234,-175.755,8.011,148.325
C09658=1219.504,400.471,-80.200,-175.755,8.009,148.325
C09659=1219.507,400.223,-80.166,-175.756,8.006,148.325
C09660=1219.511,399.975,-80.131,-175.757,8.004,148.324
C09661=1219.516,399.728,-80.097,-175.758,8.001,148.324
C09662=1219.519,399.480,-80.063,-175.758,7.999,148.323
C09663=1219.524,399.233,-80.028,-175.759,7.997,148.323
C09664=1219.528,398.985,-79.993,-175.760,7.994,148.322
C09665=1219.532,398.738,-79.959,-175.760,7.992,148.322
C09666=1219.536,398.490,-79.925,-175.761,7.990,148.321
C09667=1219.539,398.242,-79.891,-175.761,7.987,148.321
C09668=1219.544,397.995,-79.856,-175.762,7.985,148.321
C09669=1219.549,397.747,-79.822,-175.763,7.982,148.320
C09670=1219.552,397.500,-79.788,-175.763,7.980,148.320
C09671=1219.556,397.252,-79.753,-175.765,7.977,148.319
C09672=1219.560,397.004,-79.719,-175.765,7.975,148.319
C09673=1219.564,396.757,-79.684,-175.765,7.973,148.318
C09674=1219.569,396.510,-79.650,-175.766,7.970,148.318
C09675=1219.572,396.262,-79.616,-175.767,7.968,148.317
C09676=1219.576,396.014,-79.581,-175.768,7.965,148.317
C09677=1219.581,395.767,-79.548,-175.768,7.962,148.316
C09678=1219.585,395.519,-79.513,-175.769,7.960,148.316
C09679=1219.588,395.271,-79.479,-175.770,7.957,148.315
C09680=1219.593,395.024,-79.445,-175.771,7.955,148.315
C09681=1219.596,394.776,-79.411,-175.771,7.953,148.315
C09682=1219.601,394.529,-79.376,-175.772,7.949,148.314
C09683=1219.605,394.281,-79.341,-175.773,7.947,148.314
C09684=1219.609,394.033,-79.308,-175.774,7.944,148.313
C09685=1219.613,393.786,-79.274,-175.774,7.942,148.313
C09686=1219.617,393.538,-79.240,-175.775,7.940,148.312
C09687=1219.622,393.256,-79.200,-175.776,7.936,148.312
C09688=1219.626,392.974,-79.162,-175.777,7.934,148.312
C09689=1219.631,392.692,-79.122,-175.777,7.931,148.311
C09690=1219.635,392.411,-79.084,-175.778,7.928,148.310
C09691=1219.640,392.163,-79.050,-175.779,7.925,148.310
C09692=1219.643,391.915,-79.016,-175.780,7.923,148.310
C09693=1219.648,391.668,-78.981,-175.781,7.920,148.309
C09694=1219.652,391.420,-78.948,-175.782,7.918,148.309
C09695=1219.656,391.172,-78.913,-175.783,7.916,148.308
C09696=1219.660,390.925,-78.879,-175.783,7.912,148.308
C09697=1219.664,390.677,-78.845,-175.784,7.910,148.307
C09698=1219.668,390.430,-78.812,-175.785,7.908,148.307
C09699=1219.672,390.182,-78.777,-175.785,7.905,148.306
C09700=1219.676,389.935,-78.743,-175.787,7.903,148.306
C09701=1219.680,389.687,-78.709,-175.788,7.900,148.306
C09702=1219.684,389.439,-78.675,-175.788,7.897,148.305
C09703=1219.688,389.192,-78.641,-175.789,7.895,148.305
C09704=1219.693,388.944,-78.607,-175.790,7.892,148.304
C09705=1219.696,388.696,-78.573,-175.791,7.890,148.304
C09706=1219.701,388.448,-78.539,-175.792,7.887,148.303
C09707=1219.705,388.201,-78.505,-175.793,7.884,148.303
C09708=1219.709,387.953,-78.471,-175.793,7.882,148.303
C09709=1219.713,387.705,-78.437,-175.794,7.879,148.302
C09710=1219.717,387.458,-78.403,-175.795,7.876,148.302
C09711=1219.721,387.210,-78.369,-175.796,7.874,148.301
C09712=1219.725,386.962,-78.335,-175.797,7.871,148.301
C09713=1219.729,386.715,-78.300,-175.798,7.868,148.300
C09714=1219.733,386.467,-78.267,-175.799,7.866,148.300
C09715=1219.737,386.220,-78.233,-175.800,7.863,148.300
C09716=1219.741,385.971,-78.199,-175.801,7.861,148.299
C09717=1219.745,385.724,-78.165,-175.802,7.857,148.298
C09718=1219.750,385.477,-78.131,-175.802,7.855,148.298
C09719=1219.754,385.229,-78.098,-175.804,7.853,148.298
C09720=1219.757,384.981,-78.064,-175.805,7.850,148.297
C09721=1219.762,384.733,-78.030,-175.805,7.848,148.297
C09722=1219.766,384.486,-77.996,-175.806,7.845,148.296
C09723=1219.770,384.238,-77.963,-175.807,7.842,148.296
C09724=1219.774,383.990,-77.928,-175.808,7.839,148.296
C09725=1219.778,383.743,-77.895,-175.809,7.837,148.295
C09726=1219.782,383.495,-77.861,-175.810,7.834,148.295
C09727=1219.787,383.248,-77.826,-175.811,7.831,148.294
C09728=1219.791,383.000,-77.793,-175.812,7.828,148.294
C09729=1219.794,382.753,-77.759,-175.813,7.826,148.294
C09730=1219.799,382.504,-77.725,-175.814,7.824,148.293
C09731=1219.803,382.257,-77.691,-175.815,7.821,148.293
C09732=1219.807,382.010,-77.658,-175.816,7.818,148.292
C09733=1219.812,381.762,-77.625,-175.817,7.815,148.292
C09734=1219.815,381.514,-77.590,-175.818,7.812,148.291
C09735=1219.819,381.266,-77.557,-175.819,7.809,148.291
C09736=1219.823,381.019,-77.523,-175.820,7.807,148.291
C09737=1219.828,380.771,-77.490,-175.821,7.804,148.290
C09738=1219.832,380.524,-77.456,-175.822,7.802,148.290
C09739=1219.835,380.275,-77.422,-175.824,7.799,148.289
C09740=1219.840,380.027,-77.388,-175.825,7.796,148.289
C09741=1219.844,379.780,-77.355,-175.826,7.793,148.289
C09742=1219.848,379.533,-77.321,-175.827,7.790,148.288
C09743=1219.852,379.285,-77.288,-175.828,7.788,148.288
C09744=1219.856,379.037,-77.253,-175.829,7.785,148.287
C09745=1219.860,378.789,-77.220,-175.830,7.782,148.287
C09746=1219.864,378.542,-77.186,-175.831,7.780,148.287
C09747=1219.868,378.294,-77.153,-175.832,7.777,148.286
C09748=1219.873,378.046,-77.119,-175.833,7.774,148.286
C09749=1219.877,377.799,-77.086,-175.834,7.771,148.285
C09750=1219.880,377.551,-77.052,-175.836,7.768,148.285
C09751=1219.885,377.303,-77.019,-175.837,7.765,148.285
C09752=1219.888,377.056,-76.985,-175.838,7.763,148.284
C09753=1219.893,376.808,-76.951,-175.839,7.761,148.284
C09754=1219.897,376.560,-76.918,-175.840,7.758,148.283
C09755=1219.901,376.313,-76.884,-175.841,7.755,148.283
C09756=1219.905,376.065,-76.851,-175.842,7.752,148.283
C09757=1219.909,375.817,-76.818,-175.844,7.750,148.282
C09758=1219.913,375.569,-76.784,-175.845,7.747,148.282
C09759=1219.918,375.321,-76.750,-175.846,7.744,148.282
C09760=1219.922,375.074,-76.717,-175.847,7.741,148.281
C09761=1219.926,374.826,-76.684,-175.849,7.738,148.281
C09762=1219.930,374.578,-76.650,-175.850,7.736,148.280
C09763=1219.934,374.331,-76.617,-175.851,7.733,148.280
C09764=1219.938,374.083,-76.583,-175.852,7.730,148.280
C09765=1219.942,373.835,-76.550,-175.853,7.727,148.279
C09766=1219.946,373.587,-76.516,-175.854,7.724,148.279
C09767=1219.951,373.339,-76.483,-175.856,7.721,148.279
C09768=1219.955,373.092,-76.450,-175.857,7.719,148.278
C09769=1219.959,372.844,-76.416,-175.858,7.716,148.278
C09770=1219.963,372.597,-76.383,-175.860,7.713,148.278
C09771=1219.967,372.349,-76.350,-175.861,7.711,148.277
C09772=1219.971,372.101,-76.317,-175.862,7.708,148.277
C09773=1219.975,371.854,-76.283,-175.863,7.705,148.276
C09774=1219.979,371.606,-76.250,-175.865,7.702,148.276
C09775=1219.983,371.358,-76.217,-175.867,7.699,148.276
C09776=1219.988,371.110,-76.184,-175.868,7.696,148.275
C09777=1219.991,370.862,-76.149,-175.869,7.693,148.275
C09778=1219.996,370.614,-76.116,-175.870,7.690,148.275
C09779=1220.000,370.367,-76.083,-175.872,7.688,148.274
C09780=1220.004,370.119,-76.050,-175.873,7.685,148.274
C09781=1220.008,369.871,-76.016,-175.874,7.682,148.274
C09782=1220.012,369.624,-75.983,-175.875,7.679,148.273
C09783=1220.016,369.376,-75.950,-175.877,7.677,148.273
C09784=1220.020,369.128,-75.917,-175.878,7.674,148.273
C09785=1220.025,368.880,-75.884,-175.880,7.670,148.272
C09786=1220.029,368.633,-75.851,-175.882,7.668,148.272
C09787=1220.033,368.385,-75.818,-175.883,7.665,148.272
C09788=1220.037,368.137,-75.784,-175.884,7.662,148.271
C09789=1220.041,367.889,-75.751,-175.886,7.660,148.271
C09790=1220.045,367.642,-75.718,-175.887,7.657,148.271
C09791=1220.050,367.362,-75.681,-175.888,7.653,148.270
C09792=1220.055,367.082,-75.644,-175.890,7.650,148.270
C09793=1220.059,366.802,-75.606,-175.892,7.647,148.269
C09794=1220.063,366.522,-75.568,-175.893,7.644,148.269
C09795=1220.068,366.274,-75.535,-175.895,7.640,148.269
C09796=1220.072,366.026,-75.503,-175.896,7.638,148.268
C09797=1220.076,365.778,-75.470,-175.898,7.635,148.268
C09798=1220.080,365.531,-75.436,-175.899,7.633,148.268
C09799=1220.084,365.283,-75.403,-175.900,7.630,148.267
C09800=1220.089,365.035,-75.370,-175.902,7.627,148.267
C09801=1220.092,364.788,-75.338,-175.904,7.624,148.267
C09802=1220.096,364.540,-75.304,-175.905,7.621,148.266
C09803=1220.100,364.292,-75.272,-175.907,7.618,148.266
C09804=1220.105,364.044,-75.239,-175.908,7.615,148.266
C09805=1220.109,363.796,-75.206,-175.910,7.612,148.266
C09806=1220.113,363.548,-75.172,-175.911,7.609,148.265
C09807=1220.117,363.301,-75.139,-175.913,7.607,148.265
C09808=1220.122,363.053,-75.107,-175.914,7.604,148.265
C09809=1220.125,362.806,-75.075,-175.916,7.601,148.264
C09810=1220.130,362.558,-75.042,-175.917,7.598,148.264
C09811=1220.134,362.310,-75.008,-175.919,7.595,148.264
C09812=1220.138,362.062,-74.975,-175.920,7.592,148.263
C09813=1220.142,361.814,-74.943,-175.922,7.590,148.263
C09814=1220.146,361.566,-74.910,-175.924,7.586,148.263
C09815=1220.150,361.319,-74.877,-175.925,7.584,148.263
C09816=1220.154,361.071,-74.845,-175.927,7.581,148.262
C09817=1220.158,360.823,-74.811,-175.928,7.578,148.262
C09818=1220.163,360.575,-74.778,-175.930,7.575,148.262
C09819=1220.167,360.327,-74.746,-175.932,7.572,148.262
C09820=1220.170,360.079,-74.713,-175.933,7.570,148.261
C09821=1220.175,359.832,-74.680,-175.935,7.567,148.261
C09822=1220.179,359.583,-74.648,-175.936,7.563,148.261
C09823=1220.184,359.336,-74.615,-175.938,7.561,148.260
C09824=1220.188,359.088,-74.582,-175.940,7.558,148.260
C09825=1220.192,358.840,-74.550,-175.941,7.556,148.260
C09826=1220.196,358.593,-74.517,-175.943,7.552,148.260
C09827=1220.200,358.344,-74.484,-175.945,7.550,148.259
C09828=1220.204,358.097,-74.451,-175.946,7.547,148.259
C09829=1220.208,357.849,-74.419,-175.948,7.544,148.259
C09830=1220.212,357.601,-74.386,-175.950,7.541,148.259
C09831=1220.216,357.353,-74.353,-175.951,7.538,148.258
C09832=1220.221,357.106,-74.322,-175.952,7.536,148.258
C09833=1220.225,356.858,-74.288,-175.955,7.532,148.258
C09834=1220.229,356.610,-74.256,-175.956,7.530,148.258
C09835=1220.233,356.362,-74.223,-175.957,7.527,148.257
C09836=1220.237,356.114,-74.191,-175.960,7.524,148.257
C09837=1220.241,355.866,-74.158,-175.961,7.521,148.257
C09838=1220.246,355.619,-74.126,-175.963,7.519,148.257
C09839=1220.250,355.371,-74.093,-175.965,7.515,148.256
C09840=1220.254,355.123,-74.061,-175.966,7.512,148.256
C09841=1220.258,354.875,-74.028,-175.968,7.510,148.256
C09842=1220.262,354.627,-73.996,-175.970,7.506,148.256
C09843=1220.266,354.379,-73.963,-175.972,7.504,148.255
C09844=1220.270,354.132,-73.931,-175.973,7.501,148.255
C09845=1220.275,353.884,-73.899,-175.974,7.499,148.255
C09846=1220.279,353.636,-73.865,-175.977,7.495,148.255
C09847=1220.283,353.388,-73.834,-175.978,7.493,148.254
C09848=1220.287,353.140,-73.800,-175.980,7.490,148.254
C09849=1220.292,352.892,-73.768,-175.982,7.487,148.254
C09850=1220.296,352.644,-73.737,-175.984,7.484,148.254
C09851=1220.300,352.397,-73.703,-175.985,7.481,148.253
C09852=1220.303,352.149,-73.672,-175.987,7.478,148.253
C09853=1220.308,351.900,-73.639,-175.989,7.476,148.253
C09854=1220.312,351.654,-73.607,-175.990,7.473,148.253
C09855=1220.316,351.405,-73.574,-175.993,7.470,148.253
C09856=1220.321,351.157,-73.542,-175.994,7.467,148.252
C09857=1220.324,350.909,-73.510,-175.996,7.465,148.252
C09858=1220.329,350.662,-73.477,-175.998,7.461,148.252
C09859=1220.333,350.414,-73.446,-176.000,7.459,148.252
C09860=1220.337,350.165,-73.413,-176.001,7.456,148.252
C09861=1220.341,349.917,-73.381,-176.004,7.453,148.251
C09862=1220.346,349.670,-73.348,-176.005,7.450,148.251
C09863=1220.349,349.422,-73.317,-176.007,7.447,148.251
C09864=1220.354,349.174,-73.284,-176.009,7.445,148.251
C09865=1220.358,348.926,-73.252,-176.011,7.442,148.251
C09866=1220.363,348.678,-73.220,-176.013,7.439,148.250
C09867=1220.366,348.431,-73.188,-176.014,7.436,148.250
C09868=1220.371,348.183,-73.155,-176.016,7.434,148.250
C09869=1220.374,347.934,-73.123,-176.018,7.430,148.250
C09870=1220.379,347.687,-73.091,-176.020,7.428,148.250
C09871=1220.383,347.439,-73.059,-176.022,7.425,148.249
C09872=1220.387,347.190,-73.027,-176.024,7.422,148.249
C09873=1220.392,346.943,-72.996,-176.025,7.419,148.249
C09874=1220.395,346.695,-72.964,-176.027,7.417,148.249
C09875=1220.400,346.447,-72.931,-176.029,7.413,148.249
C09876=1220.404,346.200,-72.899,-176.031,7.411,148.248
C09877=1220.408,345.952,-72.867,-176.033,7.408,148.248
C09878=1220.412,345.704,-72.835,-176.035,7.405,148.248
C09879=1220.417,345.456,-72.803,-176.036,7.403,148.248
C09880=1220.421,345.208,-72.771,-176.039,7.399,148.248
C09881=1220.424,344.960,-72.739,-176.040,7.397,148.247
C09882=1220.430,344.712,-72.707,-176.042,7.394,148.247
C09883=1220.433,344.464,-72.675,-176.044,7.391,148.247
C09884=1220.437,344.216,-72.643,-176.046,7.389,148.247
C09885=1220.442,343.969,-72.611,-176.048,7.385,148.247
C09886=1220.446,343.720,-72.579,-176.050,7.383,148.247
C09887=1220.450,343.472,-72.547,-176.052,7.380,148.247
C09888=1220.454,343.225,-72.515,-176.054,7.377,148.246
C09889=1220.458,342.977,-72.484,-176.055,7.374,148.246
C09890=1220.463,342.728,-72.452,-176.058,7.371,148.246
C09891=1220.467,342.480,-72.420,-176.060,7.369,148.246
C09892=1220.471,342.232,-72.389,-176.061,7.366,148.246
C09893=1220.475,341.985,-72.357,-176.063,7.363,148.245
C09894=1220.480,341.737,-72.325,-176.065,7.360,148.245
C09895=1220.484,341.459,-72.289,-176.067,7.357,148.245
C09896=1220.489,341.181,-72.254,-176.070,7.354,148.245
C09897=1220.494,340.903,-72.218,-176.072,7.351,148.245
C09898=1220.498,340.626,-72.182,-176.074,7.348,148.245
C09899=1220.502,340.378,-72.150,-176.076,7.345,148.244
C09900=1220.507,340.129,-72.119,-176.078,7.342,148.244
C09901=1220.511,339.881,-72.087,-176.080,7.340,148.244
C09902=1220.515,339.634,-72.056,-176.082,7.336,148.244
C09903=1220.519,339.386,-72.024,-176.084,7.334,148.244
C09904=1220.524,339.138,-71.993,-176.086,7.331,148.244
C09905=1220.528,338.890,-71.961,-176.088,7.328,148.244
C09906=1220.532,338.642,-71.929,-176.089,7.326,148.244
C09907=1220.536,338.394,-71.897,-176.092,7.323,148.244
C09908=1220.540,338.146,-71.866,-176.094,7.320,148.243
C09909=1220.545,337.898,-71.834,-176.096,7.317,148.243
C09910=1220.549,337.650,-71.802,-176.098,7.314,148.243
C09911=1220.553,337.402,-71.772,-176.100,7.312,148.243
C09912=1220.557,337.154,-71.740,-176.102,7.309,148.243
C09913=1220.561,336.907,-71.708,-176.104,7.306,148.243
C09914=1220.565,336.658,-71.677,-176.106,7.303,148.243
C09915=1220.570,336.410,-71.645,-176.108,7.301,148.242
C09916=1220.574,336.162,-71.613,-176.109,7.298,148.242
C09917=1220.578,335.914,-71.582,-176.112,7.295,148.242
C09918=1220.582,335.666,-71.551,-176.114,7.293,148.242
C09919=1220.586,335.418,-71.519,-176.116,7.290,148.242
C09920=1220.591,335.170,-71.488,-176.118,7.287,148.242
C09921=1220.594,334.922,-71.456,-176.120,7.284,148.242
C09922=1220.599,334.674,-71.425,-176.122,7.281,148.242
C09923=1220.603,334.426,-71.394,-176.124,7.279,148.241
C09924=1220.607,334.178,-71.363,-176.126,7.276,148.241
C09925=1220.612,333.930,-71.330,-176.128,7.273,148.241
C09926=1220.616,333.682,-71.300,-176.130,7.270,148.241
C09927=1220.621,333.435,-71.268,-176.133,7.268,148.241
C09928=1220.625,333.186,-71.237,-176.134,7.265,148.241
C09929=1220.629,332.939,-71.205,-176.137,7.262,148.241
C09930=1220.633,332.690,-71.174,-176.138,7.260,148.241
C09931=1220.637,332.443,-71.143,-176.141,7.256,148.241
C09932=1220.641,332.194,-71.112,-176.143,7.254,148.241
C09933=1220.646,331.947,-71.080,-176.145,7.251,148.240
C09934=1220.650,331.698,-71.049,-176.147,7.249,148.240
C09935=1220.654,331.451,-71.018,-176.149,7.246,148.240
C09936=1220.658,331.202,-70.987,-176.151,7.243,148.240
C09937=1220.663,330.954,-70.956,-176.153,7.240,148.240
C09938=1220.667,330.707,-70.924,-176.156,7.237,148.240
C09939=1220.671,330.458,-70.893,-176.157,7.235,148.240
C09940=1220.675,330.210,-70.862,-176.159,7.233,148.240
C09941=1220.679,329.962,-70.831,-176.162,7.229,148.240
C09942=1220.684,329.714,-70.800,-176.164,7.227,148.240
C09943=1220.688,329.466,-70.769,-176.166,7.224,148.239
C09944=1220.691,329.218,-70.738,-176.168,7.221,148.240
C09945=1220.696,328.970,-70.707,-176.170,7.218,148.239
C09946=1220.700,328.722,-70.676,-176.172,7.216,148.239
C09947=1220.704,328.474,-70.644,-176.174,7.213,148.239
C09948=1220.709,328.226,-70.614,-176.177,7.210,148.239
C09949=1220.713,327.978,-70.582,-176.179,7.208,148.239
C09950=1220.718,327.730,-70.552,-176.181,7.205,148.239
C09951=1220.721,327.482,-70.520,-176.183,7.203,148.239
C09952=1220.726,327.234,-70.489,-176.185,7.200,148.239
C09953=1220.730,326.986,-70.458,-176.187,7.197,148.239
C09954=1220.734,326.738,-70.428,-176.189,7.194,148.239
C09955=1220.738,326.490,-70.397,-176.192,7.191,148.239
C09956=1220.743,326.242,-70.366,-176.194,7.189,148.239
C09957=1220.747,325.994,-70.334,-176.196,7.186,148.238
C09958=1220.751,325.746,-70.304,-176.198,7.184,148.239
C09959=1220.756,325.498,-70.273,-176.200,7.181,148.238
C09960=1220.759,325.249,-70.242,-176.202,7.178,148.238
C09961=1220.764,325.001,-70.212,-176.204,7.176,148.238
C09962=1220.768,324.753,-70.181,-176.207,7.172,148.238
C09963=1220.772,324.505,-70.149,-176.209,7.170,148.238
C09964=1220.776,324.258,-70.119,-176.211,7.167,148.238
C09965=1220.781,324.010,-70.088,-176.213,7.165,148.238
C09966=1220.785,323.761,-70.057,-176.215,7.162,148.238
C09967=1220.789,323.513,-70.026,-176.218,7.159,148.238
C09968=1220.793,323.265,-69.996,-176.219,7.157,148.238
C09969=1220.797,323.017,-69.965,-176.222,7.154,148.238
C09970=1220.802,322.769,-69.934,-176.224,7.152,148.238
C09971=1220.806,322.521,-69.903,-176.226,7.149,148.238
C09972=1220.810,322.273,-69.873,-176.228,7.146,148.238
C09973=1220.814,322.025,-69.842,-176.231,7.144,148.238
C09974=1220.819,321.777,-69.811,-176.233,7.140,148.238
C09975=1220.823,321.529,-69.781,-176.235,7.138,148.238
C09976=1220.827,321.280,-69.750,-176.238,7.135,148.238
C09977=1220.831,321.032,-69.719,-176.239,7.133,148.237
C09978=1220.836,320.784,-69.688,-176.241,7.130,148.238
C09979=1220.840,320.537,-69.658,-176.244,7.127,148.238
C09980=1220.844,320.287,-69.628,-176.246,7.125,148.238
C09981=1220.849,320.040,-69.597,-176.248,7.122,148.237
C09982=1220.853,319.792,-69.567,-176.250,7.120,148.237
C09983=1220.857,319.544,-69.536,-176.253,7.117,148.237
C09984=1220.861,319.296,-69.506,-176.255,7.114,148.237
C09985=1220.865,319.048,-69.475,-176.257,7.112,148.237
C09986=1220.870,318.800,-69.444,-176.259,7.109,148.237
C09987=1220.874,318.551,-69.415,-176.262,7.107,148.237
C09988=1220.879,318.303,-69.384,-176.264,7.103,148.237
C09989=1220.883,318.055,-69.353,-176.266,7.101,148.237
C09990=1220.886,317.807,-69.323,-176.268,7.099,148.237
C09991=1220.891,317.559,-69.292,-176.271,7.096,148.237
C09992=1220.895,317.311,-69.262,-176.273,7.093,148.237
C09993=1220.900,317.063,-69.232,-176.275,7.090,148.237
C09994=1220.903,316.815,-69.201,-176.277,7.088,148.237
C09995=1220.908,316.567,-69.170,-176.280,7.085,148.237
C09996=1220.912,316.318,-69.141,-176.282,7.083,148.237
//INST
///DATE 2021/06/15 17:22
///ATTR SC,RW,RJ
////FRAME ROBOT
///GROUP1 RB1
NOP
MOVL C00000 V=800.0 PL=0
MOVL C00001 V=800.0 PL=0
MOVL C00002 V=800.0 PL=0
MOVL C00003 V=800.0 PL=0
MOVL C00004 V=800.0 PL=0
MOVL C00005 V=800.0 PL=0
MOVL C00006 V=800.0 PL=0
MOVL C00007 V=800.0 PL=0
MOVL C00008 V=800.0 PL=0
MOVL C00009 V=800.0 PL=0
MOVL C00010 V=800.0 PL=0
MOVL C00011 V=800.0 PL=0
MOVL C00012 V=800.0 PL=0
MOVL C00013 V=800.0 PL=0
MOVL C00014 V=800.0 PL=0
MOVL C00015 V=800.0 PL=0
MOVL C00016 V=800.0 PL=0
MOVL C00017 V=800.0 PL=0
MOVL C00018 V=800.0 PL=0
MOVL C00019 V=800.0 PL=0
MOVL C00020 V=800.0 PL=0
MOVL C00021 V=800.0 PL=0
MOVL C00022 V=800.0 PL=0
MOVL C00023 V=800.0 PL=0
MOVL C00024 V=800.0 PL=0
MOVL C00025 V=800.0 PL=0
MOVL C00026 V=800.0 PL=0
MOVL C00027 V=800.0 PL=0
MOVL C00028 V=800.0 PL=0
MOVL C00029 V=800.0 PL=0
MOVL C00030 V=800.0 PL=0
MOVL C00031 V=800.0 PL=0
MOVL C00032 V=800.0 PL=0
MOVL C00033 V=800.0 PL=0
MOVL C00034 V=800.0 PL=0
MOVL C00035 V=800.0 PL=0
MOVL C00036 V=800.0 PL=0
MOVL C00037 V=800.0 PL=0
MOVL C00038 V=800.0 PL=0
MOVL C00039 V=800.0 PL=0
MOVL C00040 V=800.0 PL=0
MOVL C00041 V=800.0 PL=0
MOVL C00042 V=800.0 PL=0
MOVL C00043 V=800.0 PL=0
MOVL C00044 V=800.0 PL=0
MOVL C00045 V=800.0 PL=0
MOVL C00046 V=800.0 PL=0
MOVL C00047 V=800.0 PL=0
MOVL C00048 V=800.0 PL=0
MOVL C00049 V=800.0 PL=0
MOVL C00050 V=800.0 PL=0
MOVL C00051 V=800.0 PL=0
MOVL C00052 V=800.0 PL=0
MOVL C00053 V=800.0 PL=0
MOVL C00054 V=800.0 PL=0
MOVL C00055 V=800.0 PL=0
MOVL C00056 V=800.0 PL=0
MOVL C00057 V=800.0 PL=0
MOVL C00058 V=800.0 PL=0
MOVL C00059 V=800.0 PL=0
MOVL C00060 V=800.0 PL=0
MOVL C00061 V=800.0 PL=0
MOVL C00062 V=800.0 PL=0
MOVL C00063 V=800.0 PL=0
MOVL C00064 V=800.0 PL=0
MOVL C00065 V=800.0 PL=0
MOVL C00066 V=800.0 PL=0
MOVL C00067 V=800.0 PL=0
MOVL C00068 V=800.0 PL=0
MOVL C00069 V=800.0 PL=0
MOVL C00070 V=800.0 PL=0
MOVL C00071 V=800.0 PL=0
MOVL C00072 V=800.0 PL=0
MOVL C00073 V=800.0 PL=0
MOVL C00074 V=800.0 PL=0
MOVL C00075 V=800.0 PL=0
MOVL C00076 V=800.0 PL=0
MOVL C00077 V=800.0 PL=0
MOVL C00078 V=800.0 PL=0
MOVL C00079 V=800.0 PL=0
MOVL C00080 V=800.0 PL=0
MOVL C00081 V=800.0 PL=0
MOVL C00082 V=800.0 PL=0
MOVL C00083 V=800.0 PL=0
MOVL C00084 V=800.0 PL=0
MOVL C00085 V=800.0 PL=0
MOVL C00086 V=800.0 PL=0
MOVL C00087 V=800.0 PL=0
MOVL C00088 V=800.0 PL=0
MOVL C00089 V=800.0 PL=0
MOVL C00090 V=800.0 PL=0
MOVL C00091 V=800.0 PL=0
MOVL C00092 V=800.0 PL=0
MOVL C00093 V=800.0 PL=0
MOVL C00094 V=800.0 PL=0
MOVL C00095 V=800.0 PL=0
MOVL C00096 V=800.0 PL=0
MOVL C00097 V=800.0 PL=0
MOVL C00098 V=800.0 PL=0
MOVL C00099 V=800.0 PL=0
MOVL C00100 V=800.0 PL=0
MOVL C00101 V=800.0 PL=0
MOVL C00102 V=800.0 PL=0
MOVL C00103 V=800.0 PL=0
MOVL C00104 V=800.0 PL=0
MOVL C00105 V=800.0 PL=0
MOVL C00106 V=800.0 PL=0
MOVL C00107 V=800.0 PL=0
MOVL C00108 V=800.0 PL=0
MOVL C00109 V=800.0 PL=0
MOVL C00110 V=800.0 PL=0
MOVL C00111 V=800.0 PL=0
MOVL C00112 V=800.0 PL=0
MOVL C00113 V=800.0 PL=0
MOVL C00114 V=800.0 PL=0
MOVL C00115 V=800.0 PL=0
MOVL C00116 V=800.0 PL=0
MOVL C00117 V=800.0 PL=0
MOVL C00118 V=800.0 PL=0
MOVL C00119 V=800.0 PL=0
MOVL C00120 V=800.0 PL=0
MOVL C00121 V=800.0 PL=0
MOVL C00122 V=800.0 PL=0
MOVL C00123 V=800.0 PL=0
MOVL C00124 V=800.0 PL=0
MOVL C00125 V=800.0 PL=0
MOVL C00126 V=800.0 PL=0
MOVL C00127 V=800.0 PL=0
MOVL C00128 V=800.0 PL=0
MOVL C00129 V=800.0 PL=0
MOVL C00130 V=800.0 PL=0
MOVL C00131 V=800.0 PL=0
MOVL C00132 V=800.0 PL=0
MOVL C00133 V=800.0 PL=0
MOVL C00134 V=800.0 PL=0
MOVL C00135 V=800.0 PL=0
MOVL C00136 V=800.0 PL=0
MOVL C00137 V=800.0 PL=0
MOVL C00138 V=800.0 PL=0
MOVL C00139 V=800.0 PL=0
MOVL C00140 V=800.0 PL=0
MOVL C00141 V=800.0 PL=0
MOVL C00142 V=800.0 PL=0
MOVL C00143 V=800.0 PL=0
MOVL C00144 V=800.0 PL=0
MOVL C00145 V=800.0 PL=0
MOVL C00146 V=800.0 PL=0
MOVL C00147 V=800.0 PL=0
MOVL C00148 V=800.0 PL=0
MOVL C00149 V=800.0 PL=0
MOVL C00150 V=800.0 PL=0
MOVL C00151 V=800.0 PL=0
MOVL C00152 V=800.0 PL=0
MOVL C00153 V=800.0 PL=0
MOVL C00154 V=800.0 PL=0
MOVL C00155 V=800.0 PL=0
MOVL C00156 V=800.0 PL=0
MOVL C00157 V=800.0 PL=0
MOVL C00158 V=800.0 PL=0
MOVL C00159 V=800.0 PL=0
MOVL C00160 V=800.0 PL=0
MOVL C00161 V=800.0 PL=0
MOVL C00162 V=800.0 PL=0
MOVL C00163 V=800.0 PL=0
MOVL C00164 V=800.0 PL=0
MOVL C00165 V=800.0 PL=0
MOVL C00166 V=800.0 PL=0
MOVL C00167 V=800.0 PL=0
MOVL C00168 V=800.0 PL=0
MOVL C00169 V=800.0 PL=0
MOVL C00170 V=800.0 PL=0
MOVL C00171 V=800.0 PL=0
MOVL C00172 V=800.0 PL=0
MOVL C00173 V=800.0 PL=0
MOVL C00174 V=800.0 PL=0
MOVL C00175 V=800.0 PL=0
MOVL C00176 V=800.0 PL=0
MOVL C00177 V=800.0 PL=0
MOVL C00178 V=800.0 PL=0
MOVL C00179 V=800.0 PL=0
MOVL C00180 V=800.0 PL=0
MOVL C00181 V=800.0 PL=0
MOVL C00182 V=800.0 PL=0
MOVL C00183 V=800.0 PL=0
MOVL C00184 V=800.0 PL=0
MOVL C00185 V=800.0 PL=0
MOVL C00186 V=800.0 PL=0
MOVL C00187 V=800.0 PL=0
MOVL C00188 V=800.0 PL=0
MOVL C00189 V=800.0 PL=0
MOVL C00190 V=800.0 PL=0
MOVL C00191 V=800.0 PL=0
MOVL C00192 V=800.0 PL=0
MOVL C00193 V=800.0 PL=0
MOVL C00194 V=800.0 PL=0
MOVL C00195 V=800.0 PL=0
MOVL C00196 V=800.0 PL=0
MOVL C00197 V=800.0 PL=0
MOVL C00198 V=800.0 PL=0
MOVL C00199 V=800.0 PL=0
MOVL C00200 V=800.0 PL=0
MOVL C00201 V=800.0 PL=0
MOVL C00202 V=800.0 PL=0
MOVL C00203 V=800.0 PL=0
MOVL C00204 V=800.0 PL=0
MOVL C00205 V=800.0 PL=0
MOVL C00206 V=800.0 PL=0
MOVL C00207 V=800.0 PL=0
MOVL C00208 V=800.0 PL=0
MOVL C00209 V=800.0 PL=0
MOVL C00210 V=800.0 PL=0
MOVL C00211 V=800.0 PL=0
MOVL C00212 V=800.0 PL=0
MOVL C00213 V=800.0 PL=0
MOVL C00214 V=800.0 PL=0
MOVL C00215 V=800.0 PL=0
MOVL C00216 V=800.0 PL=0
MOVL C00217 V=800.0 PL=0
MOVL C00218 V=800.0 PL=0
MOVL C00219 V=800.0 PL=0
MOVL C00220 V=800.0 PL=0
MOVL C00221 V=800.0 PL=0
MOVL C00222 V=800.0 PL=0
MOVL C00223 V=800.0 PL=0
MOVL C00224 V=800.0 PL=0
MOVL C00225 V=800.0 PL=0
MOVL C00226 V=800.0 PL=0
MOVL C00227 V=800.0 PL=0
MOVL C00228 V=800.0 PL=0
MOVL C00229 V=800.0 PL=0
MOVL C00230 V=800.0 PL=0
MOVL C00231 V=800.0 PL=0
MOVL C00232 V=800.0 PL=0
MOVL C00233 V=800.0 PL=0
MOVL C00234 V=800.0 PL=0
MOVL C00235 V=800.0 PL=0
MOVL C00236 V=800.0 PL=0
MOVL C00237 V=800.0 PL=0
MOVL C00238 V=800.0 PL=0
MOVL C00239 V=800.0 PL=0
MOVL C00240 V=800.0 PL=0
MOVL C00241 V=800.0 PL=0
MOVL C00242 V=800.0 PL=0
MOVL C00243 V=800.0 PL=0
MOVL C00244 V=800.0 PL=0
MOVL C00245 V=800.0 PL=0
MOVL C00246 V=800.0 PL=0
MOVL C00247 V=800.0 PL=0
MOVL C00248 V=800.0 PL=0
MOVL C00249 V=800.0 PL=0
MOVL C00250 V=800.0 PL=0
MOVL C00251 V=800.0 PL=0
MOVL C00252 V=800.0 PL=0
MOVL C00253 V=800.0 PL=0
MOVL C00254 V=800.0 PL=0
MOVL C00255 V=800.0 PL=0
MOVL C00256 V=800.0 PL=0
MOVL C00257 V=800.0 PL=0
MOVL C00258 V=800.0 PL=0
MOVL C00259 V=800.0 PL=0
MOVL C00260 V=800.0 PL=0
MOVL C00261 V=800.0 PL=0
MOVL C00262 V=800.0 PL=0
MOVL C00263 V=800.0 PL=0
MOVL C00264 V=800.0 PL=0
MOVL C00265 V=800.0 PL=0
MOVL C00266 V=800.0 PL=0
MOVL C00267 V=800.0 PL=0
MOVL C00268 V=800.0 PL=0
MOVL C00269 V=800.0 PL=0
MOVL C00270 V=800.0 PL=0
MOVL C00271 V=800.0 PL=0
MOVL C00272 V=800.0 PL=0
MOVL C00273 V=800.0 PL=0
MOVL C00274 V=800.0 PL=0
MOVL C00275 V=800.0 PL=0
MOVL C00276 V=800.0 PL=0
MOVL C00277 V=800.0 PL=0
MOVL C00278 V=800.0 PL=0
MOVL C00279 V=800.0 PL=0
MOVL C00280 V=800.0 PL=0
MOVL C00281 V=800.0 PL=0
MOVL C00282 V=800.0 PL=0
MOVL C00283 V=800.0 PL=0
MOVL C00284 V=800.0 PL=0
MOVL C00285 V=800.0 PL=0
MOVL C00286 V=800.0 PL=0
MOVL C00287 V=800.0 PL=0
MOVL C00288 V=800.0 PL=0
MOVL C00289 V=800.0 PL=0
MOVL C00290 V=800.0 PL=0
MOVL C00291 V=800.0 PL=0
MOVL C00292 V=800.0 PL=0
MOVL C00293 V=800.0 PL=0
MOVL C00294 V=800.0 PL=0
MOVL C00295 V=800.0 PL=0
MOVL C00296 V=800.0 PL=0
MOVL C00297 V=800.0 PL=0
MOVL C00298 V=800.0 PL=0
MOVL C00299 V=800.0 PL=0
MOVL C00300 V=800.0 PL=0
MOVL C00301 V=800.0 PL=0
MOVL C00302 V=800.0 PL=0
MOVL C00303 V=800.0 PL=0
MOVL C00304 V=800.0 PL=0
MOVL C00305 V=800.0 PL=0
MOVL C00306 V=800.0 PL=0
MOVL C00307 V=800.0 PL=0
MOVL C00308 V=800.0 PL=0
MOVL C00309 V=800.0 PL=0
MOVL C00310 V=800.0 PL=0
MOVL C00311 V=800.0 PL=0
MOVL C00312 V=800.0 PL=0
MOVL C00313 V=800.0 PL=0
MOVL C00314 V=800.0 PL=0
MOVL C00315 V=800.0 PL=0
MOVL C00316 V=800.0 PL=0
MOVL C00317 V=800.0 PL=0
MOVL C00318 V=800.0 PL=0
MOVL C00319 V=800.0 PL=0
MOVL C00320 V=800.0 PL=0
MOVL C00321 V=800.0 PL=0
MOVL C00322 V=800.0 PL=0
MOVL C00323 V=800.0 PL=0
MOVL C00324 V=800.0 PL=0
MOVL C00325 V=800.0 PL=0
MOVL C00326 V=800.0 PL=0
MOVL C00327 V=800.0 PL=0
MOVL C00328 V=800.0 PL=0
MOVL C00329 V=800.0 PL=0
MOVL C00330 V=800.0 PL=0
MOVL C00331 V=800.0 PL=0
MOVL C00332 V=800.0 PL=0
MOVL C00333 V=800.0 PL=0
MOVL C00334 V=800.0 PL=0
MOVL C00335 V=800.0 PL=0
MOVL C00336 V=800.0 PL=0
MOVL C00337 V=800.0 PL=0
MOVL C00338 V=800.0 PL=0
MOVL C00339 V=800.0 PL=0
MOVL C00340 V=800.0 PL=0
MOVL C00341 V=800.0 PL=0
MOVL C00342 V=800.0 PL=0
MOVL C00343 V=800.0 PL=0
MOVL C00344 V=800.0 PL=0
MOVL C00345 V=800.0 PL=0
MOVL C00346 V=800.0 PL=0
MOVL C00347 V=800.0 PL=0
MOVL C00348 V=800.0 PL=0
MOVL C00349 V=800.0 PL=0
MOVL C00350 V=800.0 PL=0
MOVL C00351 V=800.0 PL=0
MOVL C00352 V=800.0 PL=0
MOVL C00353 V=800.0 PL=0
MOVL C00354 V=800.0 PL=0
MOVL C00355 V=800.0 PL=0
MOVL C00356 V=800.0 PL=0
MOVL C00357 V=800.0 PL=0
MOVL C00358 V=800.0 PL=0
MOVL C00359 V=800.0 PL=0
MOVL C00360 V=800.0 PL=0
MOVL C00361 V=800.0 PL=0
MOVL C00362 V=800.0 PL=0
MOVL C00363 V=800.0 PL=0
MOVL C00364 V=800.0 PL=0
MOVL C00365 V=800.0 PL=0
MOVL C00366 V=800.0 PL=0
MOVL C00367 V=800.0 PL=0
MOVL C00368 V=800.0 PL=0
MOVL C00369 V=800.0 PL=0
MOVL C00370 V=800.0 PL=0
MOVL C00371 V=800.0 PL=0
MOVL C00372 V=800.0 PL=0
MOVL C00373 V=800.0 PL=0
MOVL C00374 V=800.0 PL=0
MOVL C00375 V=800.0 PL=0
MOVL C00376 V=800.0 PL=0
MOVL C00377 V=800.0 PL=0
MOVL C00378 V=800.0 PL=0
MOVL C00379 V=800.0 PL=0
MOVL C00380 V=800.0 PL=0
MOVL C00381 V=800.0 PL=0
MOVL C00382 V=800.0 PL=0
MOVL C00383 V=800.0 PL=0
MOVL C00384 V=800.0 PL=0
MOVL C00385 V=800.0 PL=0
MOVL C00386 V=800.0 PL=0
MOVL C00387 V=800.0 PL=0
MOVL C00388 V=800.0 PL=0
MOVL C00389 V=800.0 PL=0
MOVL C00390 V=800.0 PL=0
MOVL C00391 V=800.0 PL=0
MOVL C00392 V=800.0 PL=0
MOVL C00393 V=800.0 PL=0
MOVL C00394 V=800.0 PL=0
MOVL C00395 V=800.0 PL=0
MOVL C00396 V=800.0 PL=0
MOVL C00397 V=800.0 PL=0
MOVL C00398 V=800.0 PL=0
MOVL C00399 V=800.0 PL=0
MOVL C00400 V=800.0 PL=0
MOVL C00401 V=800.0 PL=0
MOVL C00402 V=800.0 PL=0
MOVL C00403 V=800.0 PL=0
MOVL C00404 V=800.0 PL=0
MOVL C00405 V=800.0 PL=0
MOVL C00406 V=800.0 PL=0
MOVL C00407 V=800.0 PL=0
MOVL C00408 V=800.0 PL=0
MOVL C00409 V=800.0 PL=0
MOVL C00410 V=800.0 PL=0
MOVL C00411 V=800.0 PL=0
MOVL C00412 V=800.0 PL=0
MOVL C00413 V=800.0 PL=0
MOVL C00414 V=800.0 PL=0
MOVL C00415 V=800.0 PL=0
MOVL C00416 V=800.0 PL=0
MOVL C00417 V=800.0 PL=0
MOVL C00418 V=800.0 PL=0
MOVL C00419 V=800.0 PL=0
MOVL C00420 V=800.0 PL=0
MOVL C00421 V=800.0 PL=0
MOVL C00422 V=800.0 PL=0
MOVL C00423 V=800.0 PL=0
MOVL C00424 V=800.0 PL=0
MOVL C00425 V=800.0 PL=0
MOVL C00426 V=800.0 PL=0
MOVL C00427 V=800.0 PL=0
MOVL C00428 V=800.0 PL=0
MOVL C00429 V=800.0 PL=0
MOVL C00430 V=800.0 PL=0
MOVL C00431 V=800.0 PL=0
MOVL C00432 V=800.0 PL=0
MOVL C00433 V=800.0 PL=0
MOVL C00434 V=800.0 PL=0
MOVL C00435 V=800.0 PL=0
MOVL C00436 V=800.0 PL=0
MOVL C00437 V=800.0 PL=0
MOVL C00438 V=800.0 PL=0
MOVL C00439 V=800.0 PL=0
MOVL C00440 V=800.0 PL=0
MOVL C00441 V=800.0 PL=0
MOVL C00442 V=800.0 PL=0
MOVL C00443 V=800.0 PL=0
MOVL C00444 V=800.0 PL=0
MOVL C00445 V=800.0 PL=0
MOVL C00446 V=800.0 PL=0
MOVL C00447 V=800.0 PL=0
MOVL C00448 V=800.0 PL=0
MOVL C00449 V=800.0 PL=0
MOVL C00450 V=800.0 PL=0
MOVL C00451 V=800.0 PL=0
MOVL C00452 V=800.0 PL=0
MOVL C00453 V=800.0 PL=0
MOVL C00454 V=800.0 PL=0
MOVL C00455 V=800.0 PL=0
MOVL C00456 V=800.0 PL=0
MOVL C00457 V=800.0 PL=0
MOVL C00458 V=800.0 PL=0
MOVL C00459 V=800.0 PL=0
MOVL C00460 V=800.0 PL=0
MOVL C00461 V=800.0 PL=0
MOVL C00462 V=800.0 PL=0
MOVL C00463 V=800.0 PL=0
MOVL C00464 V=800.0 PL=0
MOVL C00465 V=800.0 PL=0
MOVL C00466 V=800.0 PL=0
MOVL C00467 V=800.0 PL=0
MOVL C00468 V=800.0 PL=0
MOVL C00469 V=800.0 PL=0
MOVL C00470 V=800.0 PL=0
MOVL C00471 V=800.0 PL=0
MOVL C00472 V=800.0 PL=0
MOVL C00473 V=800.0 PL=0
MOVL C00474 V=800.0 PL=0
MOVL C00475 V=800.0 PL=0
MOVL C00476 V=800.0 PL=0
MOVL C00477 V=800.0 PL=0
MOVL C00478 V=800.0 PL=0
MOVL C00479 V=800.0 PL=0
MOVL C00480 V=800.0 PL=0
MOVL C00481 V=800.0 PL=0
MOVL C00482 V=800.0 PL=0
MOVL C00483 V=800.0 PL=0
MOVL C00484 V=800.0 PL=0
MOVL C00485 V=800.0 PL=0
MOVL C00486 V=800.0 PL=0
MOVL C00487 V=800.0 PL=0
MOVL C00488 V=800.0 PL=0
MOVL C00489 V=800.0 PL=0
MOVL C00490 V=800.0 PL=0
MOVL C00491 V=800.0 PL=0
MOVL C00492 V=800.0 PL=0
MOVL C00493 V=800.0 PL=0
MOVL C00494 V=800.0 PL=0
MOVL C00495 V=800.0 PL=0
MOVL C00496 V=800.0 PL=0
MOVL C00497 V=800.0 PL=0
MOVL C00498 V=800.0 PL=0
MOVL C00499 V=800.0 PL=0
MOVL C00500 V=800.0 PL=0
MOVL C00501 V=800.0 PL=0
MOVL C00502 V=800.0 PL=0
MOVL C00503 V=800.0 PL=0
MOVL C00504 V=800.0 PL=0
MOVL C00505 V=800.0 PL=0
MOVL C00506 V=800.0 PL=0
MOVL C00507 V=800.0 PL=0
MOVL C00508 V=800.0 PL=0
MOVL C00509 V=800.0 PL=0
MOVL C00510 V=800.0 PL=0
MOVL C00511 V=800.0 PL=0
MOVL C00512 V=800.0 PL=0
MOVL C00513 V=800.0 PL=0
MOVL C00514 V=800.0 PL=0
MOVL C00515 V=800.0 PL=0
MOVL C00516 V=800.0 PL=0
MOVL C00517 V=800.0 PL=0
MOVL C00518 V=800.0 PL=0
MOVL C00519 V=800.0 PL=0
MOVL C00520 V=800.0 PL=0
MOVL C00521 V=800.0 PL=0
MOVL C00522 V=800.0 PL=0
MOVL C00523 V=800.0 PL=0
MOVL C00524 V=800.0 PL=0
MOVL C00525 V=800.0 PL=0
MOVL C00526 V=800.0 PL=0
MOVL C00527 V=800.0 PL=0
MOVL C00528 V=800.0 PL=0
MOVL C00529 V=800.0 PL=0
MOVL C00530 V=800.0 PL=0
MOVL C00531 V=800.0 PL=0
MOVL C00532 V=800.0 PL=0
MOVL C00533 V=800.0 PL=0
MOVL C00534 V=800.0 PL=0
MOVL C00535 V=800.0 PL=0
MOVL C00536 V=800.0 PL=0
MOVL C00537 V=800.0 PL=0
MOVL C00538 V=800.0 PL=0
MOVL C00539 V=800.0 PL=0
MOVL C00540 V=800.0 PL=0
MOVL C00541 V=800.0 PL=0
MOVL C00542 V=800.0 PL=0
MOVL C00543 V=800.0 PL=0
MOVL C00544 V=800.0 PL=0
MOVL C00545 V=800.0 PL=0
MOVL C00546 V=800.0 PL=0
MOVL C00547 V=800.0 PL=0
MOVL C00548 V=800.0 PL=0
MOVL C00549 V=800.0 PL=0
MOVL C00550 V=800.0 PL=0
MOVL C00551 V=800.0 PL=0
MOVL C00552 V=800.0 PL=0
MOVL C00553 V=800.0 PL=0
MOVL C00554 V=800.0 PL=0
MOVL C00555 V=800.0 PL=0
MOVL C00556 V=800.0 PL=0
MOVL C00557 V=800.0 PL=0
MOVL C00558 V=800.0 PL=0
MOVL C00559 V=800.0 PL=0
MOVL C00560 V=800.0 PL=0
MOVL C00561 V=800.0 PL=0
MOVL C00562 V=800.0 PL=0
MOVL C00563 V=800.0 PL=0
MOVL C00564 V=800.0 PL=0
MOVL C00565 V=800.0 PL=0
MOVL C00566 V=800.0 PL=0
MOVL C00567 V=800.0 PL=0
MOVL C00568 V=800.0 PL=0
MOVL C00569 V=800.0 PL=0
MOVL C00570 V=800.0 PL=0
MOVL C00571 V=800.0 PL=0
MOVL C00572 V=800.0 PL=0
MOVL C00573 V=800.0 PL=0
MOVL C00574 V=800.0 PL=0
MOVL C00575 V=800.0 PL=0
MOVL C00576 V=800.0 PL=0
MOVL C00577 V=800.0 PL=0
MOVL C00578 V=800.0 PL=0
MOVL C00579 V=800.0 PL=0
MOVL C00580 V=800.0 PL=0
MOVL C00581 V=800.0 PL=0
MOVL C00582 V=800.0 PL=0
MOVL C00583 V=800.0 PL=0
MOVL C00584 V=800.0 PL=0
MOVL C00585 V=800.0 PL=0
MOVL C00586 V=800.0 PL=0
MOVL C00587 V=800.0 PL=0
MOVL C00588 V=800.0 PL=0
MOVL C00589 V=800.0 PL=0
MOVL C00590 V=800.0 PL=0
MOVL C00591 V=800.0 PL=0
MOVL C00592 V=800.0 PL=0
MOVL C00593 V=800.0 PL=0
MOVL C00594 V=800.0 PL=0
MOVL C00595 V=800.0 PL=0
MOVL C00596 V=800.0 PL=0
MOVL C00597 V=800.0 PL=0
MOVL C00598 V=800.0 PL=0
MOVL C00599 V=800.0 PL=0
MOVL C00600 V=800.0 PL=0
MOVL C00601 V=800.0 PL=0
MOVL C00602 V=800.0 PL=0
MOVL C00603 V=800.0 PL=0
MOVL C00604 V=800.0 PL=0
MOVL C00605 V=800.0 PL=0
MOVL C00606 V=800.0 PL=0
MOVL C00607 V=800.0 PL=0
MOVL C00608 V=800.0 PL=0
MOVL C00609 V=800.0 PL=0
MOVL C00610 V=800.0 PL=0
MOVL C00611 V=800.0 PL=0
MOVL C00612 V=800.0 PL=0
MOVL C00613 V=800.0 PL=0
MOVL C00614 V=800.0 PL=0
MOVL C00615 V=800.0 PL=0
MOVL C00616 V=800.0 PL=0
MOVL C00617 V=800.0 PL=0
MOVL C00618 V=800.0 PL=0
MOVL C00619 V=800.0 PL=0
MOVL C00620 V=800.0 PL=0
MOVL C00621 V=800.0 PL=0
MOVL C00622 V=800.0 PL=0
MOVL C00623 V=800.0 PL=0
MOVL C00624 V=800.0 PL=0
MOVL C00625 V=800.0 PL=0
MOVL C00626 V=800.0 PL=0
MOVL C00627 V=800.0 PL=0
MOVL C00628 V=800.0 PL=0
MOVL C00629 V=800.0 PL=0
MOVL C00630 V=800.0 PL=0
MOVL C00631 V=800.0 PL=0
MOVL C00632 V=800.0 PL=0
MOVL C00633 V=800.0 PL=0
MOVL C00634 V=800.0 PL=0
MOVL C00635 V=800.0 PL=0
MOVL C00636 V=800.0 PL=0
MOVL C00637 V=800.0 PL=0
MOVL C00638 V=800.0 PL=0
MOVL C00639 V=800.0 PL=0
MOVL C00640 V=800.0 PL=0
MOVL C00641 V=800.0 PL=0
MOVL C00642 V=800.0 PL=0
MOVL C00643 V=800.0 PL=0
MOVL C00644 V=800.0 PL=0
MOVL C00645 V=800.0 PL=0
MOVL C00646 V=800.0 PL=0
MOVL C00647 V=800.0 PL=0
MOVL C00648 V=800.0 PL=0
MOVL C00649 V=800.0 PL=0
MOVL C00650 V=800.0 PL=0
MOVL C00651 V=800.0 PL=0
MOVL C00652 V=800.0 PL=0
MOVL C00653 V=800.0 PL=0
MOVL C00654 V=800.0 PL=0
MOVL C00655 V=800.0 PL=0
MOVL C00656 V=800.0 PL=0
MOVL C00657 V=800.0 PL=0
MOVL C00658 V=800.0 PL=0
MOVL C00659 V=800.0 PL=0
MOVL C00660 V=800.0 PL=0
MOVL C00661 V=800.0 PL=0
MOVL C00662 V=800.0 PL=0
MOVL C00663 V=800.0 PL=0
MOVL C00664 V=800.0 PL=0
MOVL C00665 V=800.0 PL=0
MOVL C00666 V=800.0 PL=0
MOVL C00667 V=800.0 PL=0
MOVL C00668 V=800.0 PL=0
MOVL C00669 V=800.0 PL=0
MOVL C00670 V=800.0 PL=0
MOVL C00671 V=800.0 PL=0
MOVL C00672 V=800.0 PL=0
MOVL C00673 V=800.0 PL=0
MOVL C00674 V=800.0 PL=0
MOVL C00675 V=800.0 PL=0
MOVL C00676 V=800.0 PL=0
MOVL C00677 V=800.0 PL=0
MOVL C00678 V=800.0 PL=0
MOVL C00679 V=800.0 PL=0
MOVL C00680 V=800.0 PL=0
MOVL C00681 V=800.0 PL=0
MOVL C00682 V=800.0 PL=0
MOVL C00683 V=800.0 PL=0
MOVL C00684 V=800.0 PL=0
MOVL C00685 V=800.0 PL=0
MOVL C00686 V=800.0 PL=0
MOVL C00687 V=800.0 PL=0
MOVL C00688 V=800.0 PL=0
MOVL C00689 V=800.0 PL=0
MOVL C00690 V=800.0 PL=0
MOVL C00691 V=800.0 PL=0
MOVL C00692 V=800.0 PL=0
MOVL C00693 V=800.0 PL=0
MOVL C00694 V=800.0 PL=0
MOVL C00695 V=800.0 PL=0
MOVL C00696 V=800.0 PL=0
MOVL C00697 V=800.0 PL=0
MOVL C00698 V=800.0 PL=0
MOVL C00699 V=800.0 PL=0
MOVL C00700 V=800.0 PL=0
MOVL C00701 V=800.0 PL=0
MOVL C00702 V=800.0 PL=0
MOVL C00703 V=800.0 PL=0
MOVL C00704 V=800.0 PL=0
MOVL C00705 V=800.0 PL=0
MOVL C00706 V=800.0 PL=0
MOVL C00707 V=800.0 PL=0
MOVL C00708 V=800.0 PL=0
MOVL C00709 V=800.0 PL=0
MOVL C00710 V=800.0 PL=0
MOVL C00711 V=800.0 PL=0
MOVL C00712 V=800.0 PL=0
MOVL C00713 V=800.0 PL=0
MOVL C00714 V=800.0 PL=0
MOVL C00715 V=800.0 PL=0
MOVL C00716 V=800.0 PL=0
MOVL C00717 V=800.0 PL=0
MOVL C00718 V=800.0 PL=0
MOVL C00719 V=800.0 PL=0
MOVL C00720 V=800.0 PL=0
MOVL C00721 V=800.0 PL=0
MOVL C00722 V=800.0 PL=0
MOVL C00723 V=800.0 PL=0
MOVL C00724 V=800.0 PL=0
MOVL C00725 V=800.0 PL=0
MOVL C00726 V=800.0 PL=0
MOVL C00727 V=800.0 PL=0
MOVL C00728 V=800.0 PL=0
MOVL C00729 V=800.0 PL=0
MOVL C00730 V=800.0 PL=0
MOVL C00731 V=800.0 PL=0
MOVL C00732 V=800.0 PL=0
MOVL C00733 V=800.0 PL=0
MOVL C00734 V=800.0 PL=0
MOVL C00735 V=800.0 PL=0
MOVL C00736 V=800.0 PL=0
MOVL C00737 V=800.0 PL=0
MOVL C00738 V=800.0 PL=0
MOVL C00739 V=800.0 PL=0
MOVL C00740 V=800.0 PL=0
MOVL C00741 V=800.0 PL=0
MOVL C00742 V=800.0 PL=0
MOVL C00743 V=800.0 PL=0
MOVL C00744 V=800.0 PL=0
MOVL C00745 V=800.0 PL=0
MOVL C00746 V=800.0 PL=0
MOVL C00747 V=800.0 PL=0
MOVL C00748 V=800.0 PL=0
MOVL C00749 V=800.0 PL=0
MOVL C00750 V=800.0 PL=0
MOVL C00751 V=800.0 PL=0
MOVL C00752 V=800.0 PL=0
MOVL C00753 V=800.0 PL=0
MOVL C00754 V=800.0 PL=0
MOVL C00755 V=800.0 PL=0
MOVL C00756 V=800.0 PL=0
MOVL C00757 V=800.0 PL=0
MOVL C00758 V=800.0 PL=0
MOVL C00759 V=800.0 PL=0
MOVL C00760 V=800.0 PL=0
MOVL C00761 V=800.0 PL=0
MOVL C00762 V=800.0 PL=0
MOVL C00763 V=800.0 PL=0
MOVL C00764 V=800.0 PL=0
MOVL C00765 V=800.0 PL=0
MOVL C00766 V=800.0 PL=0
MOVL C00767 V=800.0 PL=0
MOVL C00768 V=800.0 PL=0
MOVL C00769 V=800.0 PL=0
MOVL C00770 V=800.0 PL=0
MOVL C00771 V=800.0 PL=0
MOVL C00772 V=800.0 PL=0
MOVL C00773 V=800.0 PL=0
MOVL C00774 V=800.0 PL=0
MOVL C00775 V=800.0 PL=0
MOVL C00776 V=800.0 PL=0
MOVL C00777 V=800.0 PL=0
MOVL C00778 V=800.0 PL=0
MOVL C00779 V=800.0 PL=0
MOVL C00780 V=800.0 PL=0
MOVL C00781 V=800.0 PL=0
MOVL C00782 V=800.0 PL=0
MOVL C00783 V=800.0 PL=0
MOVL C00784 V=800.0 PL=0
MOVL C00785 V=800.0 PL=0
MOVL C00786 V=800.0 PL=0
MOVL C00787 V=800.0 PL=0
MOVL C00788 V=800.0 PL=0
MOVL C00789 V=800.0 PL=0
MOVL C00790 V=800.0 PL=0
MOVL C00791 V=800.0 PL=0
MOVL C00792 V=800.0 PL=0
MOVL C00793 V=800.0 PL=0
MOVL C00794 V=800.0 PL=0
MOVL C00795 V=800.0 PL=0
MOVL C00796 V=800.0 PL=0
MOVL C00797 V=800.0 PL=0
MOVL C00798 V=800.0 PL=0
MOVL C00799 V=800.0 PL=0
MOVL C00800 V=800.0 PL=0
MOVL C00801 V=800.0 PL=0
MOVL C00802 V=800.0 PL=0
MOVL C00803 V=800.0 PL=0
MOVL C00804 V=800.0 PL=0
MOVL C00805 V=800.0 PL=0
MOVL C00806 V=800.0 PL=0
MOVL C00807 V=800.0 PL=0
MOVL C00808 V=800.0 PL=0
MOVL C00809 V=800.0 PL=0
MOVL C00810 V=800.0 PL=0
MOVL C00811 V=800.0 PL=0
MOVL C00812 V=800.0 PL=0
MOVL C00813 V=800.0 PL=0
MOVL C00814 V=800.0 PL=0
MOVL C00815 V=800.0 PL=0
MOVL C00816 V=800.0 PL=0
MOVL C00817 V=800.0 PL=0
MOVL C00818 V=800.0 PL=0
MOVL C00819 V=800.0 PL=0
MOVL C00820 V=800.0 PL=0
MOVL C00821 V=800.0 PL=0
MOVL C00822 V=800.0 PL=0
MOVL C00823 V=800.0 PL=0
MOVL C00824 V=800.0 PL=0
MOVL C00825 V=800.0 PL=0
MOVL C00826 V=800.0 PL=0
MOVL C00827 V=800.0 PL=0
MOVL C00828 V=800.0 PL=0
MOVL C00829 V=800.0 PL=0
MOVL C00830 V=800.0 PL=0
MOVL C00831 V=800.0 PL=0
MOVL C00832 V=800.0 PL=0
MOVL C00833 V=800.0 PL=0
MOVL C00834 V=800.0 PL=0
MOVL C00835 V=800.0 PL=0
MOVL C00836 V=800.0 PL=0
MOVL C00837 V=800.0 PL=0
MOVL C00838 V=800.0 PL=0
MOVL C00839 V=800.0 PL=0
MOVL C00840 V=800.0 PL=0
MOVL C00841 V=800.0 PL=0
MOVL C00842 V=800.0 PL=0
MOVL C00843 V=800.0 PL=0
MOVL C00844 V=800.0 PL=0
MOVL C00845 V=800.0 PL=0
MOVL C00846 V=800.0 PL=0
MOVL C00847 V=800.0 PL=0
MOVL C00848 V=800.0 PL=0
MOVL C00849 V=800.0 PL=0
MOVL C00850 V=800.0 PL=0
MOVL C00851 V=800.0 PL=0
MOVL C00852 V=800.0 PL=0
MOVL C00853 V=800.0 PL=0
MOVL C00854 V=800.0 PL=0
MOVL C00855 V=800.0 PL=0
MOVL C00856 V=800.0 PL=0
MOVL C00857 V=800.0 PL=0
MOVL C00858 V=800.0 PL=0
MOVL C00859 V=800.0 PL=0
MOVL C00860 V=800.0 PL=0
MOVL C00861 V=800.0 PL=0
MOVL C00862 V=800.0 PL=0
MOVL C00863 V=800.0 PL=0
MOVL C00864 V=800.0 PL=0
MOVL C00865 V=800.0 PL=0
MOVL C00866 V=800.0 PL=0
MOVL C00867 V=800.0 PL=0
MOVL C00868 V=800.0 PL=0
MOVL C00869 V=800.0 PL=0
MOVL C00870 V=800.0 PL=0
MOVL C00871 V=800.0 PL=0
MOVL C00872 V=800.0 PL=0
MOVL C00873 V=800.0 PL=0
MOVL C00874 V=800.0 PL=0
MOVL C00875 V=800.0 PL=0
MOVL C00876 V=800.0 PL=0
MOVL C00877 V=800.0 PL=0
MOVL C00878 V=800.0 PL=0
MOVL C00879 V=800.0 PL=0
MOVL C00880 V=800.0 PL=0
MOVL C00881 V=800.0 PL=0
MOVL C00882 V=800.0 PL=0
MOVL C00883 V=800.0 PL=0
MOVL C00884 V=800.0 PL=0
MOVL C00885 V=800.0 PL=0
MOVL C00886 V=800.0 PL=0
MOVL C00887 V=800.0 PL=0
MOVL C00888 V=800.0 PL=0
MOVL C00889 V=800.0 PL=0
MOVL C00890 V=800.0 PL=0
MOVL C00891 V=800.0 PL=0
MOVL C00892 V=800.0 PL=0
MOVL C00893 V=800.0 PL=0
MOVL C00894 V=800.0 PL=0
MOVL C00895 V=800.0 PL=0
MOVL C00896 V=800.0 PL=0
MOVL C00897 V=800.0 PL=0
MOVL C00898 V=800.0 PL=0
MOVL C00899 V=800.0 PL=0
MOVL C00900 V=800.0 PL=0
MOVL C00901 V=800.0 PL=0
MOVL C00902 V=800.0 PL=0
MOVL C00903 V=800.0 PL=0
MOVL C00904 V=800.0 PL=0
MOVL C00905 V=800.0 PL=0
MOVL C00906 V=800.0 PL=0
MOVL C00907 V=800.0 PL=0
MOVL C00908 V=800.0 PL=0
MOVL C00909 V=800.0 PL=0
MOVL C00910 V=800.0 PL=0
MOVL C00911 V=800.0 PL=0
MOVL C00912 V=800.0 PL=0
MOVL C00913 V=800.0 PL=0
MOVL C00914 V=800.0 PL=0
MOVL C00915 V=800.0 PL=0
MOVL C00916 V=800.0 PL=0
MOVL C00917 V=800.0 PL=0
MOVL C00918 V=800.0 PL=0
MOVL C00919 V=800.0 PL=0
MOVL C00920 V=800.0 PL=0
MOVL C00921 V=800.0 PL=0
MOVL C00922 V=800.0 PL=0
MOVL C00923 V=800.0 PL=0
MOVL C00924 V=800.0 PL=0
MOVL C00925 V=800.0 PL=0
MOVL C00926 V=800.0 PL=0
MOVL C00927 V=800.0 PL=0
MOVL C00928 V=800.0 PL=0
MOVL C00929 V=800.0 PL=0
MOVL C00930 V=800.0 PL=0
MOVL C00931 V=800.0 PL=0
MOVL C00932 V=800.0 PL=0
MOVL C00933 V=800.0 PL=0
MOVL C00934 V=800.0 PL=0
MOVL C00935 V=800.0 PL=0
MOVL C00936 V=800.0 PL=0
MOVL C00937 V=800.0 PL=0
MOVL C00938 V=800.0 PL=0
MOVL C00939 V=800.0 PL=0
MOVL C00940 V=800.0 PL=0
MOVL C00941 V=800.0 PL=0
MOVL C00942 V=800.0 PL=0
MOVL C00943 V=800.0 PL=0
MOVL C00944 V=800.0 PL=0
MOVL C00945 V=800.0 PL=0
MOVL C00946 V=800.0 PL=0
MOVL C00947 V=800.0 PL=0
MOVL C00948 V=800.0 PL=0
MOVL C00949 V=800.0 PL=0
MOVL C00950 V=800.0 PL=0
MOVL C00951 V=800.0 PL=0
MOVL C00952 V=800.0 PL=0
MOVL C00953 V=800.0 PL=0
MOVL C00954 V=800.0 PL=0
MOVL C00955 V=800.0 PL=0
MOVL C00956 V=800.0 PL=0
MOVL C00957 V=800.0 PL=0
MOVL C00958 V=800.0 PL=0
MOVL C00959 V=800.0 PL=0
MOVL C00960 V=800.0 PL=0
MOVL C00961 V=800.0 PL=0
MOVL C00962 V=800.0 PL=0
MOVL C00963 V=800.0 PL=0
MOVL C00964 V=800.0 PL=0
MOVL C00965 V=800.0 PL=0
MOVL C00966 V=800.0 PL=0
MOVL C00967 V=800.0 PL=0
MOVL C00968 V=800.0 PL=0
MOVL C00969 V=800.0 PL=0
MOVL C00970 V=800.0 PL=0
MOVL C00971 V=800.0 PL=0
MOVL C00972 V=800.0 PL=0
MOVL C00973 V=800.0 PL=0
MOVL C00974 V=800.0 PL=0
MOVL C00975 V=800.0 PL=0
MOVL C00976 V=800.0 PL=0
MOVL C00977 V=800.0 PL=0
MOVL C00978 V=800.0 PL=0
MOVL C00979 V=800.0 PL=0
MOVL C00980 V=800.0 PL=0
MOVL C00981 V=800.0 PL=0
MOVL C00982 V=800.0 PL=0
MOVL C00983 V=800.0 PL=0
MOVL C00984 V=800.0 PL=0
MOVL C00985 V=800.0 PL=0
MOVL C00986 V=800.0 PL=0
MOVL C00987 V=800.0 PL=0
MOVL C00988 V=800.0 PL=0
MOVL C00989 V=800.0 PL=0
MOVL C00990 V=800.0 PL=0
MOVL C00991 V=800.0 PL=0
MOVL C00992 V=800.0 PL=0
MOVL C00993 V=800.0 PL=0
MOVL C00994 V=800.0 PL=0
MOVL C00995 V=800.0 PL=0
MOVL C00996 V=800.0 PL=0
MOVL C00997 V=800.0 PL=0
MOVL C00998 V=800.0 PL=0
MOVL C00999 V=800.0 PL=0
MOVL C01000 V=800.0 PL=0
MOVL C01001 V=800.0 PL=0
MOVL C01002 V=800.0 PL=0
MOVL C01003 V=800.0 PL=0
MOVL C01004 V=800.0 PL=0
MOVL C01005 V=800.0 PL=0
MOVL C01006 V=800.0 PL=0
MOVL C01007 V=800.0 PL=0
MOVL C01008 V=800.0 PL=0
MOVL C01009 V=800.0 PL=0
MOVL C01010 V=800.0 PL=0
MOVL C01011 V=800.0 PL=0
MOVL C01012 V=800.0 PL=0
MOVL C01013 V=800.0 PL=0
MOVL C01014 V=800.0 PL=0
MOVL C01015 V=800.0 PL=0
MOVL C01016 V=800.0 PL=0
MOVL C01017 V=800.0 PL=0
MOVL C01018 V=800.0 PL=0
MOVL C01019 V=800.0 PL=0
MOVL C01020 V=800.0 PL=0
MOVL C01021 V=800.0 PL=0
MOVL C01022 V=800.0 PL=0
MOVL C01023 V=800.0 PL=0
MOVL C01024 V=800.0 PL=0
MOVL C01025 V=800.0 PL=0
MOVL C01026 V=800.0 PL=0
MOVL C01027 V=800.0 PL=0
MOVL C01028 V=800.0 PL=0
MOVL C01029 V=800.0 PL=0
MOVL C01030 V=800.0 PL=0
MOVL C01031 V=800.0 PL=0
MOVL C01032 V=800.0 PL=0
MOVL C01033 V=800.0 PL=0
MOVL C01034 V=800.0 PL=0
MOVL C01035 V=800.0 PL=0
MOVL C01036 V=800.0 PL=0
MOVL C01037 V=800.0 PL=0
MOVL C01038 V=800.0 PL=0
MOVL C01039 V=800.0 PL=0
MOVL C01040 V=800.0 PL=0
MOVL C01041 V=800.0 PL=0
MOVL C01042 V=800.0 PL=0
MOVL C01043 V=800.0 PL=0
MOVL C01044 V=800.0 PL=0
MOVL C01045 V=800.0 PL=0
MOVL C01046 V=800.0 PL=0
MOVL C01047 V=800.0 PL=0
MOVL C01048 V=800.0 PL=0
MOVL C01049 V=800.0 PL=0
MOVL C01050 V=800.0 PL=0
MOVL C01051 V=800.0 PL=0
MOVL C01052 V=800.0 PL=0
MOVL C01053 V=800.0 PL=0
MOVL C01054 V=800.0 PL=0
MOVL C01055 V=800.0 PL=0
MOVL C01056 V=800.0 PL=0
MOVL C01057 V=800.0 PL=0
MOVL C01058 V=800.0 PL=0
MOVL C01059 V=800.0 PL=0
MOVL C01060 V=800.0 PL=0
MOVL C01061 V=800.0 PL=0
MOVL C01062 V=800.0 PL=0
MOVL C01063 V=800.0 PL=0
MOVL C01064 V=800.0 PL=0
MOVL C01065 V=800.0 PL=0
MOVL C01066 V=800.0 PL=0
MOVL C01067 V=800.0 PL=0
MOVL C01068 V=800.0 PL=0
MOVL C01069 V=800.0 PL=0
MOVL C01070 V=800.0 PL=0
MOVL C01071 V=800.0 PL=0
MOVL C01072 V=800.0 PL=0
MOVL C01073 V=800.0 PL=0
MOVL C01074 V=800.0 PL=0
MOVL C01075 V=800.0 PL=0
MOVL C01076 V=800.0 PL=0
MOVL C01077 V=800.0 PL=0
MOVL C01078 V=800.0 PL=0
MOVL C01079 V=800.0 PL=0
MOVL C01080 V=800.0 PL=0
MOVL C01081 V=800.0 PL=0
MOVL C01082 V=800.0 PL=0
MOVL C01083 V=800.0 PL=0
MOVL C01084 V=800.0 PL=0
MOVL C01085 V=800.0 PL=0
MOVL C01086 V=800.0 PL=0
MOVL C01087 V=800.0 PL=0
MOVL C01088 V=800.0 PL=0
MOVL C01089 V=800.0 PL=0
MOVL C01090 V=800.0 PL=0
MOVL C01091 V=800.0 PL=0
MOVL C01092 V=800.0 PL=0
MOVL C01093 V=800.0 PL=0
MOVL C01094 V=800.0 PL=0
MOVL C01095 V=800.0 PL=0
MOVL C01096 V=800.0 PL=0
MOVL C01097 V=800.0 PL=0
MOVL C01098 V=800.0 PL=0
MOVL C01099 V=800.0 PL=0
MOVL C01100 V=800.0 PL=0
MOVL C01101 V=800.0 PL=0
MOVL C01102 V=800.0 PL=0
MOVL C01103 V=800.0 PL=0
MOVL C01104 V=800.0 PL=0
MOVL C01105 V=800.0 PL=0
MOVL C01106 V=800.0 PL=0
MOVL C01107 V=800.0 PL=0
MOVL C01108 V=800.0 PL=0
MOVL C01109 V=800.0 PL=0
MOVL C01110 V=800.0 PL=0
MOVL C01111 V=800.0 PL=0
MOVL C01112 V=800.0 PL=0
MOVL C01113 V=800.0 PL=0
MOVL C01114 V=800.0 PL=0
MOVL C01115 V=800.0 PL=0
MOVL C01116 V=800.0 PL=0
MOVL C01117 V=800.0 PL=0
MOVL C01118 V=800.0 PL=0
MOVL C01119 V=800.0 PL=0
MOVL C01120 V=800.0 PL=0
MOVL C01121 V=800.0 PL=0
MOVL C01122 V=800.0 PL=0
MOVL C01123 V=800.0 PL=0
MOVL C01124 V=800.0 PL=0
MOVL C01125 V=800.0 PL=0
MOVL C01126 V=800.0 PL=0
MOVL C01127 V=800.0 PL=0
MOVL C01128 V=800.0 PL=0
MOVL C01129 V=800.0 PL=0
MOVL C01130 V=800.0 PL=0
MOVL C01131 V=800.0 PL=0
MOVL C01132 V=800.0 PL=0
MOVL C01133 V=800.0 PL=0
MOVL C01134 V=800.0 PL=0
MOVL C01135 V=800.0 PL=0
MOVL C01136 V=800.0 PL=0
MOVL C01137 V=800.0 PL=0
MOVL C01138 V=800.0 PL=0
MOVL C01139 V=800.0 PL=0
MOVL C01140 V=800.0 PL=0
MOVL C01141 V=800.0 PL=0
MOVL C01142 V=800.0 PL=0
MOVL C01143 V=800.0 PL=0
MOVL C01144 V=800.0 PL=0
MOVL C01145 V=800.0 PL=0
MOVL C01146 V=800.0 PL=0
MOVL C01147 V=800.0 PL=0
MOVL C01148 V=800.0 PL=0
MOVL C01149 V=800.0 PL=0
MOVL C01150 V=800.0 PL=0
MOVL C01151 V=800.0 PL=0
MOVL C01152 V=800.0 PL=0
MOVL C01153 V=800.0 PL=0
MOVL C01154 V=800.0 PL=0
MOVL C01155 V=800.0 PL=0
MOVL C01156 V=800.0 PL=0
MOVL C01157 V=800.0 PL=0
MOVL C01158 V=800.0 PL=0
MOVL C01159 V=800.0 PL=0
MOVL C01160 V=800.0 PL=0
MOVL C01161 V=800.0 PL=0
MOVL C01162 V=800.0 PL=0
MOVL C01163 V=800.0 PL=0
MOVL C01164 V=800.0 PL=0
MOVL C01165 V=800.0 PL=0
MOVL C01166 V=800.0 PL=0
MOVL C01167 V=800.0 PL=0
MOVL C01168 V=800.0 PL=0
MOVL C01169 V=800.0 PL=0
MOVL C01170 V=800.0 PL=0
MOVL C01171 V=800.0 PL=0
MOVL C01172 V=800.0 PL=0
MOVL C01173 V=800.0 PL=0
MOVL C01174 V=800.0 PL=0
MOVL C01175 V=800.0 PL=0
MOVL C01176 V=800.0 PL=0
MOVL C01177 V=800.0 PL=0
MOVL C01178 V=800.0 PL=0
MOVL C01179 V=800.0 PL=0
MOVL C01180 V=800.0 PL=0
MOVL C01181 V=800.0 PL=0
MOVL C01182 V=800.0 PL=0
MOVL C01183 V=800.0 PL=0
MOVL C01184 V=800.0 PL=0
MOVL C01185 V=800.0 PL=0
MOVL C01186 V=800.0 PL=0
MOVL C01187 V=800.0 PL=0
MOVL C01188 V=800.0 PL=0
MOVL C01189 V=800.0 PL=0
MOVL C01190 V=800.0 PL=0
MOVL C01191 V=800.0 PL=0
MOVL C01192 V=800.0 PL=0
MOVL C01193 V=800.0 PL=0
MOVL C01194 V=800.0 PL=0
MOVL C01195 V=800.0 PL=0
MOVL C01196 V=800.0 PL=0
MOVL C01197 V=800.0 PL=0
MOVL C01198 V=800.0 PL=0
MOVL C01199 V=800.0 PL=0
MOVL C01200 V=800.0 PL=0
MOVL C01201 V=800.0 PL=0
MOVL C01202 V=800.0 PL=0
MOVL C01203 V=800.0 PL=0
MOVL C01204 V=800.0 PL=0
MOVL C01205 V=800.0 PL=0
MOVL C01206 V=800.0 PL=0
MOVL C01207 V=800.0 PL=0
MOVL C01208 V=800.0 PL=0
MOVL C01209 V=800.0 PL=0
MOVL C01210 V=800.0 PL=0
MOVL C01211 V=800.0 PL=0
MOVL C01212 V=800.0 PL=0
MOVL C01213 V=800.0 PL=0
MOVL C01214 V=800.0 PL=0
MOVL C01215 V=800.0 PL=0
MOVL C01216 V=800.0 PL=0
MOVL C01217 V=800.0 PL=0
MOVL C01218 V=800.0 PL=0
MOVL C01219 V=800.0 PL=0
MOVL C01220 V=800.0 PL=0
MOVL C01221 V=800.0 PL=0
MOVL C01222 V=800.0 PL=0
MOVL C01223 V=800.0 PL=0
MOVL C01224 V=800.0 PL=0
MOVL C01225 V=800.0 PL=0
MOVL C01226 V=800.0 PL=0
MOVL C01227 V=800.0 PL=0
MOVL C01228 V=800.0 PL=0
MOVL C01229 V=800.0 PL=0
MOVL C01230 V=800.0 PL=0
MOVL C01231 V=800.0 PL=0
MOVL C01232 V=800.0 PL=0
MOVL C01233 V=800.0 PL=0
MOVL C01234 V=800.0 PL=0
MOVL C01235 V=800.0 PL=0
MOVL C01236 V=800.0 PL=0
MOVL C01237 V=800.0 PL=0
MOVL C01238 V=800.0 PL=0
MOVL C01239 V=800.0 PL=0
MOVL C01240 V=800.0 PL=0
MOVL C01241 V=800.0 PL=0
MOVL C01242 V=800.0 PL=0
MOVL C01243 V=800.0 PL=0
MOVL C01244 V=800.0 PL=0
MOVL C01245 V=800.0 PL=0
MOVL C01246 V=800.0 PL=0
MOVL C01247 V=800.0 PL=0
MOVL C01248 V=800.0 PL=0
MOVL C01249 V=800.0 PL=0
MOVL C01250 V=800.0 PL=0
MOVL C01251 V=800.0 PL=0
MOVL C01252 V=800.0 PL=0
MOVL C01253 V=800.0 PL=0
MOVL C01254 V=800.0 PL=0
MOVL C01255 V=800.0 PL=0
MOVL C01256 V=800.0 PL=0
MOVL C01257 V=800.0 PL=0
MOVL C01258 V=800.0 PL=0
MOVL C01259 V=800.0 PL=0
MOVL C01260 V=800.0 PL=0
MOVL C01261 V=800.0 PL=0
MOVL C01262 V=800.0 PL=0
MOVL C01263 V=800.0 PL=0
MOVL C01264 V=800.0 PL=0
MOVL C01265 V=800.0 PL=0
MOVL C01266 V=800.0 PL=0
MOVL C01267 V=800.0 PL=0
MOVL C01268 V=800.0 PL=0
MOVL C01269 V=800.0 PL=0
MOVL C01270 V=800.0 PL=0
MOVL C01271 V=800.0 PL=0
MOVL C01272 V=800.0 PL=0
MOVL C01273 V=800.0 PL=0
MOVL C01274 V=800.0 PL=0
MOVL C01275 V=800.0 PL=0
MOVL C01276 V=800.0 PL=0
MOVL C01277 V=800.0 PL=0
MOVL C01278 V=800.0 PL=0
MOVL C01279 V=800.0 PL=0
MOVL C01280 V=800.0 PL=0
MOVL C01281 V=800.0 PL=0
MOVL C01282 V=800.0 PL=0
MOVL C01283 V=800.0 PL=0
MOVL C01284 V=800.0 PL=0
MOVL C01285 V=800.0 PL=0
MOVL C01286 V=800.0 PL=0
MOVL C01287 V=800.0 PL=0
MOVL C01288 V=800.0 PL=0
MOVL C01289 V=800.0 PL=0
MOVL C01290 V=800.0 PL=0
MOVL C01291 V=800.0 PL=0
MOVL C01292 V=800.0 PL=0
MOVL C01293 V=800.0 PL=0
MOVL C01294 V=800.0 PL=0
MOVL C01295 V=800.0 PL=0
MOVL C01296 V=800.0 PL=0
MOVL C01297 V=800.0 PL=0
MOVL C01298 V=800.0 PL=0
MOVL C01299 V=800.0 PL=0
MOVL C01300 V=800.0 PL=0
MOVL C01301 V=800.0 PL=0
MOVL C01302 V=800.0 PL=0
MOVL C01303 V=800.0 PL=0
MOVL C01304 V=800.0 PL=0
MOVL C01305 V=800.0 PL=0
MOVL C01306 V=800.0 PL=0
MOVL C01307 V=800.0 PL=0
MOVL C01308 V=800.0 PL=0
MOVL C01309 V=800.0 PL=0
MOVL C01310 V=800.0 PL=0
MOVL C01311 V=800.0 PL=0
MOVL C01312 V=800.0 PL=0
MOVL C01313 V=800.0 PL=0
MOVL C01314 V=800.0 PL=0
MOVL C01315 V=800.0 PL=0
MOVL C01316 V=800.0 PL=0
MOVL C01317 V=800.0 PL=0
MOVL C01318 V=800.0 PL=0
MOVL C01319 V=800.0 PL=0
MOVL C01320 V=800.0 PL=0
MOVL C01321 V=800.0 PL=0
MOVL C01322 V=800.0 PL=0
MOVL C01323 V=800.0 PL=0
MOVL C01324 V=800.0 PL=0
MOVL C01325 V=800.0 PL=0
MOVL C01326 V=800.0 PL=0
MOVL C01327 V=800.0 PL=0
MOVL C01328 V=800.0 PL=0
MOVL C01329 V=800.0 PL=0
MOVL C01330 V=800.0 PL=0
MOVL C01331 V=800.0 PL=0
MOVL C01332 V=800.0 PL=0
MOVL C01333 V=800.0 PL=0
MOVL C01334 V=800.0 PL=0
MOVL C01335 V=800.0 PL=0
MOVL C01336 V=800.0 PL=0
MOVL C01337 V=800.0 PL=0
MOVL C01338 V=800.0 PL=0
MOVL C01339 V=800.0 PL=0
MOVL C01340 V=800.0 PL=0
MOVL C01341 V=800.0 PL=0
MOVL C01342 V=800.0 PL=0
MOVL C01343 V=800.0 PL=0
MOVL C01344 V=800.0 PL=0
MOVL C01345 V=800.0 PL=0
MOVL C01346 V=800.0 PL=0
MOVL C01347 V=800.0 PL=0
MOVL C01348 V=800.0 PL=0
MOVL C01349 V=800.0 PL=0
MOVL C01350 V=800.0 PL=0
MOVL C01351 V=800.0 PL=0
MOVL C01352 V=800.0 PL=0
MOVL C01353 V=800.0 PL=0
MOVL C01354 V=800.0 PL=0
MOVL C01355 V=800.0 PL=0
MOVL C01356 V=800.0 PL=0
MOVL C01357 V=800.0 PL=0
MOVL C01358 V=800.0 PL=0
MOVL C01359 V=800.0 PL=0
MOVL C01360 V=800.0 PL=0
MOVL C01361 V=800.0 PL=0
MOVL C01362 V=800.0 PL=0
MOVL C01363 V=800.0 PL=0
MOVL C01364 V=800.0 PL=0
MOVL C01365 V=800.0 PL=0
MOVL C01366 V=800.0 PL=0
MOVL C01367 V=800.0 PL=0
MOVL C01368 V=800.0 PL=0
MOVL C01369 V=800.0 PL=0
MOVL C01370 V=800.0 PL=0
MOVL C01371 V=800.0 PL=0
MOVL C01372 V=800.0 PL=0
MOVL C01373 V=800.0 PL=0
MOVL C01374 V=800.0 PL=0
MOVL C01375 V=800.0 PL=0
MOVL C01376 V=800.0 PL=0
MOVL C01377 V=800.0 PL=0
MOVL C01378 V=800.0 PL=0
MOVL C01379 V=800.0 PL=0
MOVL C01380 V=800.0 PL=0
MOVL C01381 V=800.0 PL=0
MOVL C01382 V=800.0 PL=0
MOVL C01383 V=800.0 PL=0
MOVL C01384 V=800.0 PL=0
MOVL C01385 V=800.0 PL=0
MOVL C01386 V=800.0 PL=0
MOVL C01387 V=800.0 PL=0
MOVL C01388 V=800.0 PL=0
MOVL C01389 V=800.0 PL=0
MOVL C01390 V=800.0 PL=0
MOVL C01391 V=800.0 PL=0
MOVL C01392 V=800.0 PL=0
MOVL C01393 V=800.0 PL=0
MOVL C01394 V=800.0 PL=0
MOVL C01395 V=800.0 PL=0
MOVL C01396 V=800.0 PL=0
MOVL C01397 V=800.0 PL=0
MOVL C01398 V=800.0 PL=0
MOVL C01399 V=800.0 PL=0
MOVL C01400 V=800.0 PL=0
MOVL C01401 V=800.0 PL=0
MOVL C01402 V=800.0 PL=0
MOVL C01403 V=800.0 PL=0
MOVL C01404 V=800.0 PL=0
MOVL C01405 V=800.0 PL=0
MOVL C01406 V=800.0 PL=0
MOVL C01407 V=800.0 PL=0
MOVL C01408 V=800.0 PL=0
MOVL C01409 V=800.0 PL=0
MOVL C01410 V=800.0 PL=0
MOVL C01411 V=800.0 PL=0
MOVL C01412 V=800.0 PL=0
MOVL C01413 V=800.0 PL=0
MOVL C01414 V=800.0 PL=0
MOVL C01415 V=800.0 PL=0
MOVL C01416 V=800.0 PL=0
MOVL C01417 V=800.0 PL=0
MOVL C01418 V=800.0 PL=0
MOVL C01419 V=800.0 PL=0
MOVL C01420 V=800.0 PL=0
MOVL C01421 V=800.0 PL=0
MOVL C01422 V=800.0 PL=0
MOVL C01423 V=800.0 PL=0
MOVL C01424 V=800.0 PL=0
MOVL C01425 V=800.0 PL=0
MOVL C01426 V=800.0 PL=0
MOVL C01427 V=800.0 PL=0
MOVL C01428 V=800.0 PL=0
MOVL C01429 V=800.0 PL=0
MOVL C01430 V=800.0 PL=0
MOVL C01431 V=800.0 PL=0
MOVL C01432 V=800.0 PL=0
MOVL C01433 V=800.0 PL=0
MOVL C01434 V=800.0 PL=0
MOVL C01435 V=800.0 PL=0
MOVL C01436 V=800.0 PL=0
MOVL C01437 V=800.0 PL=0
MOVL C01438 V=800.0 PL=0
MOVL C01439 V=800.0 PL=0
MOVL C01440 V=800.0 PL=0
MOVL C01441 V=800.0 PL=0
MOVL C01442 V=800.0 PL=0
MOVL C01443 V=800.0 PL=0
MOVL C01444 V=800.0 PL=0
MOVL C01445 V=800.0 PL=0
MOVL C01446 V=800.0 PL=0
MOVL C01447 V=800.0 PL=0
MOVL C01448 V=800.0 PL=0
MOVL C01449 V=800.0 PL=0
MOVL C01450 V=800.0 PL=0
MOVL C01451 V=800.0 PL=0
MOVL C01452 V=800.0 PL=0
MOVL C01453 V=800.0 PL=0
MOVL C01454 V=800.0 PL=0
MOVL C01455 V=800.0 PL=0
MOVL C01456 V=800.0 PL=0
MOVL C01457 V=800.0 PL=0
MOVL C01458 V=800.0 PL=0
MOVL C01459 V=800.0 PL=0
MOVL C01460 V=800.0 PL=0
MOVL C01461 V=800.0 PL=0
MOVL C01462 V=800.0 PL=0
MOVL C01463 V=800.0 PL=0
MOVL C01464 V=800.0 PL=0
MOVL C01465 V=800.0 PL=0
MOVL C01466 V=800.0 PL=0
MOVL C01467 V=800.0 PL=0
MOVL C01468 V=800.0 PL=0
MOVL C01469 V=800.0 PL=0
MOVL C01470 V=800.0 PL=0
MOVL C01471 V=800.0 PL=0
MOVL C01472 V=800.0 PL=0
MOVL C01473 V=800.0 PL=0
MOVL C01474 V=800.0 PL=0
MOVL C01475 V=800.0 PL=0
MOVL C01476 V=800.0 PL=0
MOVL C01477 V=800.0 PL=0
MOVL C01478 V=800.0 PL=0
MOVL C01479 V=800.0 PL=0
MOVL C01480 V=800.0 PL=0
MOVL C01481 V=800.0 PL=0
MOVL C01482 V=800.0 PL=0
MOVL C01483 V=800.0 PL=0
MOVL C01484 V=800.0 PL=0
MOVL C01485 V=800.0 PL=0
MOVL C01486 V=800.0 PL=0
MOVL C01487 V=800.0 PL=0
MOVL C01488 V=800.0 PL=0
MOVL C01489 V=800.0 PL=0
MOVL C01490 V=800.0 PL=0
MOVL C01491 V=800.0 PL=0
MOVL C01492 V=800.0 PL=0
MOVL C01493 V=800.0 PL=0
MOVL C01494 V=800.0 PL=0
MOVL C01495 V=800.0 PL=0
MOVL C01496 V=800.0 PL=0
MOVL C01497 V=800.0 PL=0
MOVL C01498 V=800.0 PL=0
MOVL C01499 V=800.0 PL=0
MOVL C01500 V=800.0 PL=0
MOVL C01501 V=800.0 PL=0
MOVL C01502 V=800.0 PL=0
MOVL C01503 V=800.0 PL=0
MOVL C01504 V=800.0 PL=0
MOVL C01505 V=800.0 PL=0
MOVL C01506 V=800.0 PL=0
MOVL C01507 V=800.0 PL=0
MOVL C01508 V=800.0 PL=0
MOVL C01509 V=800.0 PL=0
MOVL C01510 V=800.0 PL=0
MOVL C01511 V=800.0 PL=0
MOVL C01512 V=800.0 PL=0
MOVL C01513 V=800.0 PL=0
MOVL C01514 V=800.0 PL=0
MOVL C01515 V=800.0 PL=0
MOVL C01516 V=800.0 PL=0
MOVL C01517 V=800.0 PL=0
MOVL C01518 V=800.0 PL=0
MOVL C01519 V=800.0 PL=0
MOVL C01520 V=800.0 PL=0
MOVL C01521 V=800.0 PL=0
MOVL C01522 V=800.0 PL=0
MOVL C01523 V=800.0 PL=0
MOVL C01524 V=800.0 PL=0
MOVL C01525 V=800.0 PL=0
MOVL C01526 V=800.0 PL=0
MOVL C01527 V=800.0 PL=0
MOVL C01528 V=800.0 PL=0
MOVL C01529 V=800.0 PL=0
MOVL C01530 V=800.0 PL=0
MOVL C01531 V=800.0 PL=0
MOVL C01532 V=800.0 PL=0
MOVL C01533 V=800.0 PL=0
MOVL C01534 V=800.0 PL=0
MOVL C01535 V=800.0 PL=0
MOVL C01536 V=800.0 PL=0
MOVL C01537 V=800.0 PL=0
MOVL C01538 V=800.0 PL=0
MOVL C01539 V=800.0 PL=0
MOVL C01540 V=800.0 PL=0
MOVL C01541 V=800.0 PL=0
MOVL C01542 V=800.0 PL=0
MOVL C01543 V=800.0 PL=0
MOVL C01544 V=800.0 PL=0
MOVL C01545 V=800.0 PL=0
MOVL C01546 V=800.0 PL=0
MOVL C01547 V=800.0 PL=0
MOVL C01548 V=800.0 PL=0
MOVL C01549 V=800.0 PL=0
MOVL C01550 V=800.0 PL=0
MOVL C01551 V=800.0 PL=0
MOVL C01552 V=800.0 PL=0
MOVL C01553 V=800.0 PL=0
MOVL C01554 V=800.0 PL=0
MOVL C01555 V=800.0 PL=0
MOVL C01556 V=800.0 PL=0
MOVL C01557 V=800.0 PL=0
MOVL C01558 V=800.0 PL=0
MOVL C01559 V=800.0 PL=0
MOVL C01560 V=800.0 PL=0
MOVL C01561 V=800.0 PL=0
MOVL C01562 V=800.0 PL=0
MOVL C01563 V=800.0 PL=0
MOVL C01564 V=800.0 PL=0
MOVL C01565 V=800.0 PL=0
MOVL C01566 V=800.0 PL=0
MOVL C01567 V=800.0 PL=0
MOVL C01568 V=800.0 PL=0
MOVL C01569 V=800.0 PL=0
MOVL C01570 V=800.0 PL=0
MOVL C01571 V=800.0 PL=0
MOVL C01572 V=800.0 PL=0
MOVL C01573 V=800.0 PL=0
MOVL C01574 V=800.0 PL=0
MOVL C01575 V=800.0 PL=0
MOVL C01576 V=800.0 PL=0
MOVL C01577 V=800.0 PL=0
MOVL C01578 V=800.0 PL=0
MOVL C01579 V=800.0 PL=0
MOVL C01580 V=800.0 PL=0
MOVL C01581 V=800.0 PL=0
MOVL C01582 V=800.0 PL=0
MOVL C01583 V=800.0 PL=0
MOVL C01584 V=800.0 PL=0
MOVL C01585 V=800.0 PL=0
MOVL C01586 V=800.0 PL=0
MOVL C01587 V=800.0 PL=0
MOVL C01588 V=800.0 PL=0
MOVL C01589 V=800.0 PL=0
MOVL C01590 V=800.0 PL=0
MOVL C01591 V=800.0 PL=0
MOVL C01592 V=800.0 PL=0
MOVL C01593 V=800.0 PL=0
MOVL C01594 V=800.0 PL=0
MOVL C01595 V=800.0 PL=0
MOVL C01596 V=800.0 PL=0
MOVL C01597 V=800.0 PL=0
MOVL C01598 V=800.0 PL=0
MOVL C01599 V=800.0 PL=0
MOVL C01600 V=800.0 PL=0
MOVL C01601 V=800.0 PL=0
MOVL C01602 V=800.0 PL=0
MOVL C01603 V=800.0 PL=0
MOVL C01604 V=800.0 PL=0
MOVL C01605 V=800.0 PL=0
MOVL C01606 V=800.0 PL=0
MOVL C01607 V=800.0 PL=0
MOVL C01608 V=800.0 PL=0
MOVL C01609 V=800.0 PL=0
MOVL C01610 V=800.0 PL=0
MOVL C01611 V=800.0 PL=0
MOVL C01612 V=800.0 PL=0
MOVL C01613 V=800.0 PL=0
MOVL C01614 V=800.0 PL=0
MOVL C01615 V=800.0 PL=0
MOVL C01616 V=800.0 PL=0
MOVL C01617 V=800.0 PL=0
MOVL C01618 V=800.0 PL=0
MOVL C01619 V=800.0 PL=0
MOVL C01620 V=800.0 PL=0
MOVL C01621 V=800.0 PL=0
MOVL C01622 V=800.0 PL=0
MOVL C01623 V=800.0 PL=0
MOVL C01624 V=800.0 PL=0
MOVL C01625 V=800.0 PL=0
MOVL C01626 V=800.0 PL=0
MOVL C01627 V=800.0 PL=0
MOVL C01628 V=800.0 PL=0
MOVL C01629 V=800.0 PL=0
MOVL C01630 V=800.0 PL=0
MOVL C01631 V=800.0 PL=0
MOVL C01632 V=800.0 PL=0
MOVL C01633 V=800.0 PL=0
MOVL C01634 V=800.0 PL=0
MOVL C01635 V=800.0 PL=0
MOVL C01636 V=800.0 PL=0
MOVL C01637 V=800.0 PL=0
MOVL C01638 V=800.0 PL=0
MOVL C01639 V=800.0 PL=0
MOVL C01640 V=800.0 PL=0
MOVL C01641 V=800.0 PL=0
MOVL C01642 V=800.0 PL=0
MOVL C01643 V=800.0 PL=0
MOVL C01644 V=800.0 PL=0
MOVL C01645 V=800.0 PL=0
MOVL C01646 V=800.0 PL=0
MOVL C01647 V=800.0 PL=0
MOVL C01648 V=800.0 PL=0
MOVL C01649 V=800.0 PL=0
MOVL C01650 V=800.0 PL=0
MOVL C01651 V=800.0 PL=0
MOVL C01652 V=800.0 PL=0
MOVL C01653 V=800.0 PL=0
MOVL C01654 V=800.0 PL=0
MOVL C01655 V=800.0 PL=0
MOVL C01656 V=800.0 PL=0
MOVL C01657 V=800.0 PL=0
MOVL C01658 V=800.0 PL=0
MOVL C01659 V=800.0 PL=0
MOVL C01660 V=800.0 PL=0
MOVL C01661 V=800.0 PL=0
MOVL C01662 V=800.0 PL=0
MOVL C01663 V=800.0 PL=0
MOVL C01664 V=800.0 PL=0
MOVL C01665 V=800.0 PL=0
MOVL C01666 V=800.0 PL=0
MOVL C01667 V=800.0 PL=0
MOVL C01668 V=800.0 PL=0
MOVL C01669 V=800.0 PL=0
MOVL C01670 V=800.0 PL=0
MOVL C01671 V=800.0 PL=0
MOVL C01672 V=800.0 PL=0
MOVL C01673 V=800.0 PL=0
MOVL C01674 V=800.0 PL=0
MOVL C01675 V=800.0 PL=0
MOVL C01676 V=800.0 PL=0
MOVL C01677 V=800.0 PL=0
MOVL C01678 V=800.0 PL=0
MOVL C01679 V=800.0 PL=0
MOVL C01680 V=800.0 PL=0
MOVL C01681 V=800.0 PL=0
MOVL C01682 V=800.0 PL=0
MOVL C01683 V=800.0 PL=0
MOVL C01684 V=800.0 PL=0
MOVL C01685 V=800.0 PL=0
MOVL C01686 V=800.0 PL=0
MOVL C01687 V=800.0 PL=0
MOVL C01688 V=800.0 PL=0
MOVL C01689 V=800.0 PL=0
MOVL C01690 V=800.0 PL=0
MOVL C01691 V=800.0 PL=0
MOVL C01692 V=800.0 PL=0
MOVL C01693 V=800.0 PL=0
MOVL C01694 V=800.0 PL=0
MOVL C01695 V=800.0 PL=0
MOVL C01696 V=800.0 PL=0
MOVL C01697 V=800.0 PL=0
MOVL C01698 V=800.0 PL=0
MOVL C01699 V=800.0 PL=0
MOVL C01700 V=800.0 PL=0
MOVL C01701 V=800.0 PL=0
MOVL C01702 V=800.0 PL=0
MOVL C01703 V=800.0 PL=0
MOVL C01704 V=800.0 PL=0
MOVL C01705 V=800.0 PL=0
MOVL C01706 V=800.0 PL=0
MOVL C01707 V=800.0 PL=0
MOVL C01708 V=800.0 PL=0
MOVL C01709 V=800.0 PL=0
MOVL C01710 V=800.0 PL=0
MOVL C01711 V=800.0 PL=0
MOVL C01712 V=800.0 PL=0
MOVL C01713 V=800.0 PL=0
MOVL C01714 V=800.0 PL=0
MOVL C01715 V=800.0 PL=0
MOVL C01716 V=800.0 PL=0
MOVL C01717 V=800.0 PL=0
MOVL C01718 V=800.0 PL=0
MOVL C01719 V=800.0 PL=0
MOVL C01720 V=800.0 PL=0
MOVL C01721 V=800.0 PL=0
MOVL C01722 V=800.0 PL=0
MOVL C01723 V=800.0 PL=0
MOVL C01724 V=800.0 PL=0
MOVL C01725 V=800.0 PL=0
MOVL C01726 V=800.0 PL=0
MOVL C01727 V=800.0 PL=0
MOVL C01728 V=800.0 PL=0
MOVL C01729 V=800.0 PL=0
MOVL C01730 V=800.0 PL=0
MOVL C01731 V=800.0 PL=0
MOVL C01732 V=800.0 PL=0
MOVL C01733 V=800.0 PL=0
MOVL C01734 V=800.0 PL=0
MOVL C01735 V=800.0 PL=0
MOVL C01736 V=800.0 PL=0
MOVL C01737 V=800.0 PL=0
MOVL C01738 V=800.0 PL=0
MOVL C01739 V=800.0 PL=0
MOVL C01740 V=800.0 PL=0
MOVL C01741 V=800.0 PL=0
MOVL C01742 V=800.0 PL=0
MOVL C01743 V=800.0 PL=0
MOVL C01744 V=800.0 PL=0
MOVL C01745 V=800.0 PL=0
MOVL C01746 V=800.0 PL=0
MOVL C01747 V=800.0 PL=0
MOVL C01748 V=800.0 PL=0
MOVL C01749 V=800.0 PL=0
MOVL C01750 V=800.0 PL=0
MOVL C01751 V=800.0 PL=0
MOVL C01752 V=800.0 PL=0
MOVL C01753 V=800.0 PL=0
MOVL C01754 V=800.0 PL=0
MOVL C01755 V=800.0 PL=0
MOVL C01756 V=800.0 PL=0
MOVL C01757 V=800.0 PL=0
MOVL C01758 V=800.0 PL=0
MOVL C01759 V=800.0 PL=0
MOVL C01760 V=800.0 PL=0
MOVL C01761 V=800.0 PL=0
MOVL C01762 V=800.0 PL=0
MOVL C01763 V=800.0 PL=0
MOVL C01764 V=800.0 PL=0
MOVL C01765 V=800.0 PL=0
MOVL C01766 V=800.0 PL=0
MOVL C01767 V=800.0 PL=0
MOVL C01768 V=800.0 PL=0
MOVL C01769 V=800.0 PL=0
MOVL C01770 V=800.0 PL=0
MOVL C01771 V=800.0 PL=0
MOVL C01772 V=800.0 PL=0
MOVL C01773 V=800.0 PL=0
MOVL C01774 V=800.0 PL=0
MOVL C01775 V=800.0 PL=0
MOVL C01776 V=800.0 PL=0
MOVL C01777 V=800.0 PL=0
MOVL C01778 V=800.0 PL=0
MOVL C01779 V=800.0 PL=0
MOVL C01780 V=800.0 PL=0
MOVL C01781 V=800.0 PL=0
MOVL C01782 V=800.0 PL=0
MOVL C01783 V=800.0 PL=0
MOVL C01784 V=800.0 PL=0
MOVL C01785 V=800.0 PL=0
MOVL C01786 V=800.0 PL=0
MOVL C01787 V=800.0 PL=0
MOVL C01788 V=800.0 PL=0
MOVL C01789 V=800.0 PL=0
MOVL C01790 V=800.0 PL=0
MOVL C01791 V=800.0 PL=0
MOVL C01792 V=800.0 PL=0
MOVL C01793 V=800.0 PL=0
MOVL C01794 V=800.0 PL=0
MOVL C01795 V=800.0 PL=0
MOVL C01796 V=800.0 PL=0
MOVL C01797 V=800.0 PL=0
MOVL C01798 V=800.0 PL=0
MOVL C01799 V=800.0 PL=0
MOVL C01800 V=800.0 PL=0
MOVL C01801 V=800.0 PL=0
MOVL C01802 V=800.0 PL=0
MOVL C01803 V=800.0 PL=0
MOVL C01804 V=800.0 PL=0
MOVL C01805 V=800.0 PL=0
MOVL C01806 V=800.0 PL=0
MOVL C01807 V=800.0 PL=0
MOVL C01808 V=800.0 PL=0
MOVL C01809 V=800.0 PL=0
MOVL C01810 V=800.0 PL=0
MOVL C01811 V=800.0 PL=0
MOVL C01812 V=800.0 PL=0
MOVL C01813 V=800.0 PL=0
MOVL C01814 V=800.0 PL=0
MOVL C01815 V=800.0 PL=0
MOVL C01816 V=800.0 PL=0
MOVL C01817 V=800.0 PL=0
MOVL C01818 V=800.0 PL=0
MOVL C01819 V=800.0 PL=0
MOVL C01820 V=800.0 PL=0
MOVL C01821 V=800.0 PL=0
MOVL C01822 V=800.0 PL=0
MOVL C01823 V=800.0 PL=0
MOVL C01824 V=800.0 PL=0
MOVL C01825 V=800.0 PL=0
MOVL C01826 V=800.0 PL=0
MOVL C01827 V=800.0 PL=0
MOVL C01828 V=800.0 PL=0
MOVL C01829 V=800.0 PL=0
MOVL C01830 V=800.0 PL=0
MOVL C01831 V=800.0 PL=0
MOVL C01832 V=800.0 PL=0
MOVL C01833 V=800.0 PL=0
MOVL C01834 V=800.0 PL=0
MOVL C01835 V=800.0 PL=0
MOVL C01836 V=800.0 PL=0
MOVL C01837 V=800.0 PL=0
MOVL C01838 V=800.0 PL=0
MOVL C01839 V=800.0 PL=0
MOVL C01840 V=800.0 PL=0
MOVL C01841 V=800.0 PL=0
MOVL C01842 V=800.0 PL=0
MOVL C01843 V=800.0 PL=0
MOVL C01844 V=800.0 PL=0
MOVL C01845 V=800.0 PL=0
MOVL C01846 V=800.0 PL=0
MOVL C01847 V=800.0 PL=0
MOVL C01848 V=800.0 PL=0
MOVL C01849 V=800.0 PL=0
MOVL C01850 V=800.0 PL=0
MOVL C01851 V=800.0 PL=0
MOVL C01852 V=800.0 PL=0
MOVL C01853 V=800.0 PL=0
MOVL C01854 V=800.0 PL=0
MOVL C01855 V=800.0 PL=0
MOVL C01856 V=800.0 PL=0
MOVL C01857 V=800.0 PL=0
MOVL C01858 V=800.0 PL=0
MOVL C01859 V=800.0 PL=0
MOVL C01860 V=800.0 PL=0
MOVL C01861 V=800.0 PL=0
MOVL C01862 V=800.0 PL=0
MOVL C01863 V=800.0 PL=0
MOVL C01864 V=800.0 PL=0
MOVL C01865 V=800.0 PL=0
MOVL C01866 V=800.0 PL=0
MOVL C01867 V=800.0 PL=0
MOVL C01868 V=800.0 PL=0
MOVL C01869 V=800.0 PL=0
MOVL C01870 V=800.0 PL=0
MOVL C01871 V=800.0 PL=0
MOVL C01872 V=800.0 PL=0
MOVL C01873 V=800.0 PL=0
MOVL C01874 V=800.0 PL=0
MOVL C01875 V=800.0 PL=0
MOVL C01876 V=800.0 PL=0
MOVL C01877 V=800.0 PL=0
MOVL C01878 V=800.0 PL=0
MOVL C01879 V=800.0 PL=0
MOVL C01880 V=800.0 PL=0
MOVL C01881 V=800.0 PL=0
MOVL C01882 V=800.0 PL=0
MOVL C01883 V=800.0 PL=0
MOVL C01884 V=800.0 PL=0
MOVL C01885 V=800.0 PL=0
MOVL C01886 V=800.0 PL=0
MOVL C01887 V=800.0 PL=0
MOVL C01888 V=800.0 PL=0
MOVL C01889 V=800.0 PL=0
MOVL C01890 V=800.0 PL=0
MOVL C01891 V=800.0 PL=0
MOVL C01892 V=800.0 PL=0
MOVL C01893 V=800.0 PL=0
MOVL C01894 V=800.0 PL=0
MOVL C01895 V=800.0 PL=0
MOVL C01896 V=800.0 PL=0
MOVL C01897 V=800.0 PL=0
MOVL C01898 V=800.0 PL=0
MOVL C01899 V=800.0 PL=0
MOVL C01900 V=800.0 PL=0
MOVL C01901 V=800.0 PL=0
MOVL C01902 V=800.0 PL=0
MOVL C01903 V=800.0 PL=0
MOVL C01904 V=800.0 PL=0
MOVL C01905 V=800.0 PL=0
MOVL C01906 V=800.0 PL=0
MOVL C01907 V=800.0 PL=0
MOVL C01908 V=800.0 PL=0
MOVL C01909 V=800.0 PL=0
MOVL C01910 V=800.0 PL=0
MOVL C01911 V=800.0 PL=0
MOVL C01912 V=800.0 PL=0
MOVL C01913 V=800.0 PL=0
MOVL C01914 V=800.0 PL=0
MOVL C01915 V=800.0 PL=0
MOVL C01916 V=800.0 PL=0
MOVL C01917 V=800.0 PL=0
MOVL C01918 V=800.0 PL=0
MOVL C01919 V=800.0 PL=0
MOVL C01920 V=800.0 PL=0
MOVL C01921 V=800.0 PL=0
MOVL C01922 V=800.0 PL=0
MOVL C01923 V=800.0 PL=0
MOVL C01924 V=800.0 PL=0
MOVL C01925 V=800.0 PL=0
MOVL C01926 V=800.0 PL=0
MOVL C01927 V=800.0 PL=0
MOVL C01928 V=800.0 PL=0
MOVL C01929 V=800.0 PL=0
MOVL C01930 V=800.0 PL=0
MOVL C01931 V=800.0 PL=0
MOVL C01932 V=800.0 PL=0
MOVL C01933 V=800.0 PL=0
MOVL C01934 V=800.0 PL=0
MOVL C01935 V=800.0 PL=0
MOVL C01936 V=800.0 PL=0
MOVL C01937 V=800.0 PL=0
MOVL C01938 V=800.0 PL=0
MOVL C01939 V=800.0 PL=0
MOVL C01940 V=800.0 PL=0
MOVL C01941 V=800.0 PL=0
MOVL C01942 V=800.0 PL=0
MOVL C01943 V=800.0 PL=0
MOVL C01944 V=800.0 PL=0
MOVL C01945 V=800.0 PL=0
MOVL C01946 V=800.0 PL=0
MOVL C01947 V=800.0 PL=0
MOVL C01948 V=800.0 PL=0
MOVL C01949 V=800.0 PL=0
MOVL C01950 V=800.0 PL=0
MOVL C01951 V=800.0 PL=0
MOVL C01952 V=800.0 PL=0
MOVL C01953 V=800.0 PL=0
MOVL C01954 V=800.0 PL=0
MOVL C01955 V=800.0 PL=0
MOVL C01956 V=800.0 PL=0
MOVL C01957 V=800.0 PL=0
MOVL C01958 V=800.0 PL=0
MOVL C01959 V=800.0 PL=0
MOVL C01960 V=800.0 PL=0
MOVL C01961 V=800.0 PL=0
MOVL C01962 V=800.0 PL=0
MOVL C01963 V=800.0 PL=0
MOVL C01964 V=800.0 PL=0
MOVL C01965 V=800.0 PL=0
MOVL C01966 V=800.0 PL=0
MOVL C01967 V=800.0 PL=0
MOVL C01968 V=800.0 PL=0
MOVL C01969 V=800.0 PL=0
MOVL C01970 V=800.0 PL=0
MOVL C01971 V=800.0 PL=0
MOVL C01972 V=800.0 PL=0
MOVL C01973 V=800.0 PL=0
MOVL C01974 V=800.0 PL=0
MOVL C01975 V=800.0 PL=0
MOVL C01976 V=800.0 PL=0
MOVL C01977 V=800.0 PL=0
MOVL C01978 V=800.0 PL=0
MOVL C01979 V=800.0 PL=0
MOVL C01980 V=800.0 PL=0
MOVL C01981 V=800.0 PL=0
MOVL C01982 V=800.0 PL=0
MOVL C01983 V=800.0 PL=0
MOVL C01984 V=800.0 PL=0
MOVL C01985 V=800.0 PL=0
MOVL C01986 V=800.0 PL=0
MOVL C01987 V=800.0 PL=0
MOVL C01988 V=800.0 PL=0
MOVL C01989 V=800.0 PL=0
MOVL C01990 V=800.0 PL=0
MOVL C01991 V=800.0 PL=0
MOVL C01992 V=800.0 PL=0
MOVL C01993 V=800.0 PL=0
MOVL C01994 V=800.0 PL=0
MOVL C01995 V=800.0 PL=0
MOVL C01996 V=800.0 PL=0
MOVL C01997 V=800.0 PL=0
MOVL C01998 V=800.0 PL=0
MOVL C01999 V=800.0 PL=0
MOVL C02000 V=800.0 PL=0
MOVL C02001 V=800.0 PL=0
MOVL C02002 V=800.0 PL=0
MOVL C02003 V=800.0 PL=0
MOVL C02004 V=800.0 PL=0
MOVL C02005 V=800.0 PL=0
MOVL C02006 V=800.0 PL=0
MOVL C02007 V=800.0 PL=0
MOVL C02008 V=800.0 PL=0
MOVL C02009 V=800.0 PL=0
MOVL C02010 V=800.0 PL=0
MOVL C02011 V=800.0 PL=0
MOVL C02012 V=800.0 PL=0
MOVL C02013 V=800.0 PL=0
MOVL C02014 V=800.0 PL=0
MOVL C02015 V=800.0 PL=0
MOVL C02016 V=800.0 PL=0
MOVL C02017 V=800.0 PL=0
MOVL C02018 V=800.0 PL=0
MOVL C02019 V=800.0 PL=0
MOVL C02020 V=800.0 PL=0
MOVL C02021 V=800.0 PL=0
MOVL C02022 V=800.0 PL=0
MOVL C02023 V=800.0 PL=0
MOVL C02024 V=800.0 PL=0
MOVL C02025 V=800.0 PL=0
MOVL C02026 V=800.0 PL=0
MOVL C02027 V=800.0 PL=0
MOVL C02028 V=800.0 PL=0
MOVL C02029 V=800.0 PL=0
MOVL C02030 V=800.0 PL=0
MOVL C02031 V=800.0 PL=0
MOVL C02032 V=800.0 PL=0
MOVL C02033 V=800.0 PL=0
MOVL C02034 V=800.0 PL=0
MOVL C02035 V=800.0 PL=0
MOVL C02036 V=800.0 PL=0
MOVL C02037 V=800.0 PL=0
MOVL C02038 V=800.0 PL=0
MOVL C02039 V=800.0 PL=0
MOVL C02040 V=800.0 PL=0
MOVL C02041 V=800.0 PL=0
MOVL C02042 V=800.0 PL=0
MOVL C02043 V=800.0 PL=0
MOVL C02044 V=800.0 PL=0
MOVL C02045 V=800.0 PL=0
MOVL C02046 V=800.0 PL=0
MOVL C02047 V=800.0 PL=0
MOVL C02048 V=800.0 PL=0
MOVL C02049 V=800.0 PL=0
MOVL C02050 V=800.0 PL=0
MOVL C02051 V=800.0 PL=0
MOVL C02052 V=800.0 PL=0
MOVL C02053 V=800.0 PL=0
MOVL C02054 V=800.0 PL=0
MOVL C02055 V=800.0 PL=0
MOVL C02056 V=800.0 PL=0
MOVL C02057 V=800.0 PL=0
MOVL C02058 V=800.0 PL=0
MOVL C02059 V=800.0 PL=0
MOVL C02060 V=800.0 PL=0
MOVL C02061 V=800.0 PL=0
MOVL C02062 V=800.0 PL=0
MOVL C02063 V=800.0 PL=0
MOVL C02064 V=800.0 PL=0
MOVL C02065 V=800.0 PL=0
MOVL C02066 V=800.0 PL=0
MOVL C02067 V=800.0 PL=0
MOVL C02068 V=800.0 PL=0
MOVL C02069 V=800.0 PL=0
MOVL C02070 V=800.0 PL=0
MOVL C02071 V=800.0 PL=0
MOVL C02072 V=800.0 PL=0
MOVL C02073 V=800.0 PL=0
MOVL C02074 V=800.0 PL=0
MOVL C02075 V=800.0 PL=0
MOVL C02076 V=800.0 PL=0
MOVL C02077 V=800.0 PL=0
MOVL C02078 V=800.0 PL=0
MOVL C02079 V=800.0 PL=0
MOVL C02080 V=800.0 PL=0
MOVL C02081 V=800.0 PL=0
MOVL C02082 V=800.0 PL=0
MOVL C02083 V=800.0 PL=0
MOVL C02084 V=800.0 PL=0
MOVL C02085 V=800.0 PL=0
MOVL C02086 V=800.0 PL=0
